SPLINE
SPL {X  -134.098, Y  +772.750, Z    +0.000, E1   -45.587, E3 +302845.435}
SPL {X  -155.319, Y  +733.085, Z    +0.000, E1   -31.947, E3 +302836.313}
SPL {X  -162.077, Y  +709.719, Z    +0.000, E1   -21.590, E3 +302837.990}
SPL {X  -164.499, Y  +694.994, Z    +0.000, E1   -13.860, E3 +302838.775}
SPL {X  -165.382, Y  +684.927, Z    +0.000, E1    -7.984, E3 +302836.952}
SPL {X  -165.645, Y  +676.778, Z    +0.000, E1    -2.777, E3 +302836.675}
SPL {X  -165.650, Y  +672.041, Z    +0.000, E1    +0.844, E3 +302835.366}
SPL {X  -165.650, Y  +667.328, Z    +0.000, E1    +5.806, E3 +302834.743}
SPL {X  -165.650, Y  +661.774, Z    +0.000, E1   +13.006, E3 +302833.067}
SPL {X  -165.650, Y  +656.573, Z    +0.000, E1   +19.875, E3 +302833.626}
SPL {X  -165.650, Y  +650.769, Z    +0.000, E1   +28.083, E3 +302831.992}
SPL {X  -165.650, Y  +639.700, Z    +0.000, E1   +43.326, E3 +302827.054}
SPL {X  -165.650, Y  +605.320, Z    +0.000, E1   +76.562, E3 +302806.463}
SPL {X  -165.650, Y  +597.745, Z    +0.000, E1   +59.636, E3 +302844.464}
SPL {X  -165.650, Y  +596.360, Z    +0.000, E1   +54.978, E3 +302858.072}
SPL {X  -165.650, Y  +524.050, Z    +0.000, E1   +59.300, E3 +302919.978}
ENDSPLINE

SPLINE
SPL {X  -165.650, Y  +539.856, Z    +0.000, E1   +53.398, E3 +302935.626}
ENDSPLINE

SPLINE
SPL {X  -165.650, Y  +530.389, Z    +0.000, E1   +53.621, E3 +302948.631}
SPL {X  -165.650, Y  +521.849, Z    +0.000, E1   +53.452, E3 +302962.571}
SPL {X  -165.650, Y  +515.134, Z    +0.000, E1   +53.252, E3 +302973.922}
SPL {X  -165.650, Y  +505.685, Z    +0.000, E1   +53.701, E3 +302985.529}
SPL {X  -165.650, Y  +498.275, Z    +0.000, E1   +53.357, E3 +302998.837}
SPL {X  -165.650, Y  +491.031, Z    +0.000, E1   +53.348, E3 +303009.857}
SPL {X  -165.650, Y  +479.077, Z    +0.000, E1   +55.039, E3 +303016.980}
SPL {X  -165.650, Y  +450.615, Z    +0.000, E1   +59.721, E3 +303023.486}
SPL {X  -165.650, Y  +449.326, Z    +0.000, E1   +58.606, E3 +303032.535}
SPL {X  -165.650, Y  +442.154, Z    +0.000, E1   +58.369, E3 +303043.159}
SPL {X  -165.650, Y  +437.405, Z    +0.000, E1   +57.663, E3 +303053.769}
SPL {X  -165.650, Y  +432.227, Z    +0.000, E1   +57.103, E3 +303064.256}
SPL {X  -165.650, Y  +428.683, Z    +0.000, E1   +56.222, E3 +303074.611}
SPL {X  -165.650, Y  +424.202, Z    +0.000, E1   +55.382, E3 +303086.300}
SPL {X  -165.650, Y  +418.756, Z    +0.000, E1   +54.154, E3 +303101.979}
SPL {X  -165.650, Y  +407.872, Z    +0.000, E1   +54.003, E3 +303119.064}
SPL {X  -165.650, Y  +400.791, Z    +0.000, E1   +53.827, E3 +303130.507}
SPL {X  -165.650, Y  +393.046, Z    +0.000, E1   +53.951, E3 +303141.399}
SPL {X  -165.650, Y  +383.306, Z    +0.000, E1   +53.987, E3 +303155.676}
SPL {X  -165.640, Y  +376.676, Z    +0.000, E1   +53.760, E3 +303166.843}
SPL {X  -165.408, Y  +369.556, Z    +0.000, E1   +53.942, E3 +303176.394}
SPL {X  -164.927, Y  +363.041, Z    +0.000, E1   +53.687, E3 +303187.690}
SPL {X  -164.096, Y  +355.862, Z    +0.000, E1   +53.838, E3 +303197.420}
SPL {X  -162.936, Y  +348.637, Z    +0.000, E1   +53.390, E3 +303211.136}
SPL {X  -161.218, Y  +340.437, Z    +0.000, E1   +53.207, E3 +303224.248}
SPL {X  -159.523, Y  +333.864, Z    +0.000, E1   +52.908, E3 +303235.870}
SPL {X  -157.624, Y  +327.563, Z    +0.000, E1   +52.705, E3 +303246.280}
SPL {X  -155.665, Y  +321.859, Z    +0.000, E1   +52.064, E3 +303258.453}
SPL {X  -152.682, Y  +314.249, Z    +0.000, E1   +51.841, E3 +303270.901}
SPL {X  -150.607, Y  +309.525, Z    +0.000, E1   +51.147, E3 +303281.385}
SPL {X  -142.104, Y  +293.374, Z    +0.000, E1   +55.775, E3 +303281.117}
SPL {X  -134.755, Y  +282.163, Z    +0.000, E1   +57.236, E3 +303287.385}
SPL {X  -117.053, Y  +261.289, Z    +0.000, E1   +49.815, E3 +303396.897}
ENDSPLINE

SPLINE
SPL {X  -148.836, Y  +305.783, Z    +0.000, E1   +38.029, E3 +303488.375}
SPL {X  -161.816, Y  +343.065, Z    +0.000, E1   +22.147, E3 +303479.025}
SPL {X  -164.614, Y  +360.007, Z    +0.000, E1   +13.213, E3 +303474.811}
SPL {X  -165.520, Y  +371.933, Z    +0.000, E1    +6.276, E3 +303477.565}
SPL {X  -165.650, Y  +378.704, Z    +0.000, E1    +1.700, E3 +303476.435}
SPL {X  -165.650, Y  +382.197, Z    +0.000, E1    -1.038, E3 +303475.508}
SPL {X  -165.650, Y  +386.782, Z    +0.000, E1    -5.783, E3 +303474.986}
SPL {X  -165.650, Y  +392.406, Z    +0.000, E1   -13.042, E3 +303472.883}
SPL {X  -165.650, Y  +398.038, Z    +0.000, E1   -20.113, E3 +303474.450}
SPL {X  -165.650, Y  +403.005, Z    +0.000, E1   -26.762, E3 +303473.632}
SPL {X  -165.650, Y  +415.469, Z    +0.000, E1   -43.461, E3 +303468.455}
SPL {X  -165.650, Y  +460.095, Z    +0.000, E1   -60.221, E3 +303486.717}
SPL {X  -165.650, Y  +535.749, Z    +0.000, E1   -60.559, E3 +303557.560}
ENDSPLINE

SPLINE
SPL {X  -165.650, Y  +516.750, Z    +0.000, E1   -54.244, E3 +303573.411}
ENDSPLINE

SPLINE
SPL {X  -165.650, Y  +524.345, Z    +0.000, E1   -54.115, E3 +303585.308}
SPL {X  -165.650, Y  +531.171, Z    +0.000, E1   -54.075, E3 +303595.746}
SPL {X  -165.650, Y  +538.771, Z    +0.000, E1   -53.840, E3 +303608.486}
SPL {X  -165.650, Y  +548.103, Z    +0.000, E1   -53.944, E3 +303621.833}
SPL {X  -165.650, Y  +558.071, Z    +0.000, E1   -53.870, E3 +303637.174}
SPL {X  -165.650, Y  +568.053, Z    +0.000, E1   -54.124, E3 +303650.351}
SPL {X  -165.650, Y  +577.021, Z    +0.000, E1   -53.813, E3 +303665.850}
SPL {X  -165.650, Y  +587.996, Z    +0.000, E1   -53.969, E3 +303681.088}
SPL {X  -165.650, Y  +595.185, Z    +0.000, E1   -53.962, E3 +303691.797}
SPL {X  -165.650, Y  +602.138, Z    +0.000, E1   -53.941, E3 +303702.291}
SPL {X  -165.650, Y  +610.307, Z    +0.000, E1   -53.995, E3 +303714.139}
SPL {X  -165.650, Y  +617.878, Z    +0.000, E1   -53.838, E3 +303726.396}
SPL {X  -165.650, Y  +626.374, Z    +0.000, E1   -54.092, E3 +303737.411}
SPL {X  -165.650, Y  +632.964, Z    +0.000, E1   -53.887, E3 +303748.539}
SPL {X  -165.650, Y  +640.262, Z    +0.000, E1   -53.965, E3 +303758.853}
SPL {X  -165.650, Y  +647.911, Z    +0.000, E1   -53.930, E3 +303770.608}
SPL {X  -165.650, Y  +658.189, Z    +0.000, E1   -53.932, E3 +303785.908}
SPL {X  -165.650, Y  +667.820, Z    +0.000, E1   -53.975, E3 +303799.934}
SPL {X  -165.623, Y  +678.503, Z    +0.000, E1   -53.932, E3 +303816.286}
SPL {X  -165.171, Y  +688.090, Z    +0.000, E1   -54.025, E3 +303829.734}
SPL {X  -164.558, Y  +694.489, Z    +0.000, E1   -53.745, E3 +303841.083}
SPL {X  -163.580, Y  +701.606, Z    +0.000, E1   -53.591, E3 +303852.516}
SPL {X  -162.702, Y  +706.614, Z    +0.000, E1   -53.230, E3 +303862.183}
SPL {X  -160.941, Y  +714.715, Z    +0.000, E1   -53.321, E3 +303873.802}
SPL {X  -159.638, Y  +719.723, Z    +0.000, E1   -52.685, E3 +303884.805}
SPL {X  -157.521, Y  +726.754, Z    +0.000, E1   -52.585, E3 +303896.000}
SPL {X  -155.632, Y  +732.234, Z    +0.000, E1   -52.209, E3 +303906.047}
SPL {X  -153.975, Y  +736.588, Z    +0.000, E1   -51.877, E3 +303914.373}
SPL {X  -151.949, Y  +741.465, Z    +0.000, E1   -51.645, E3 +303922.779}
SPL {X  -149.075, Y  +747.727, Z    +0.000, E1   -52.134, E3 +303929.493}
SPL {X  -137.775, Y  +767.467, Z    +0.000, E1   -56.912, E3 +303932.157}
SPL {X  -128.847, Y  +779.607, Z    +0.000, E1   -49.118, E3 +304007.173}
SPL {X   -94.133, Y  +811.804, Z    +0.000, E1   -53.019, E3 +304061.807}
ENDSPLINE

SPLINE
SPL {X  -123.886, Y  +785.464, Z    +0.000, E1   -49.465, E3 +304146.834}
SPL {X  -152.385, Y  +740.452, Z    +0.000, E1   -34.821, E3 +304127.811}
SPL {X  -162.077, Y  +709.719, Z    +0.000, E1   -21.590, E3 +304129.657}
SPL {X  -164.499, Y  +694.994, Z    +0.000, E1   -13.860, E3 +304130.442}
SPL {X  -165.382, Y  +684.927, Z    +0.000, E1    -7.984, E3 +304128.619}
SPL {X  -165.645, Y  +676.778, Z    +0.000, E1    -2.777, E3 +304128.341}
SPL {X  -165.650, Y  +672.041, Z    +0.000, E1    +0.844, E3 +304127.033}
SPL {X  -165.650, Y  +667.328, Z    +0.000, E1    +5.806, E3 +304126.410}
SPL {X  -165.650, Y  +661.774, Z    +0.000, E1   +13.006, E3 +304124.734}
SPL {X  -165.650, Y  +654.085, Z    +0.000, E1   +23.232, E3 +304124.593}
SPL {X  -165.650, Y  +639.700, Z    +0.000, E1   +43.326, E3 +304118.720}
SPL {X  -165.650, Y  +605.320, Z    +0.000, E1   +76.562, E3 +304098.130}
SPL {X  -165.650, Y  +597.745, Z    +0.000, E1   +59.636, E3 +304136.131}
SPL {X  -165.650, Y  +596.360, Z    +0.000, E1   +54.978, E3 +304149.739}
SPL {X  -165.650, Y  +524.050, Z    +0.000, E1   +59.300, E3 +304211.645}
ENDSPLINE

SPLINE
SPL {X  -165.650, Y  +539.856, Z    +0.000, E1   +53.398, E3 +304227.292}
ENDSPLINE

SPLINE
SPL {X  -165.650, Y  +530.389, Z    +0.000, E1   +53.621, E3 +304240.298}
SPL {X  -165.650, Y  +521.849, Z    +0.000, E1   +53.452, E3 +304254.237}
SPL {X  -165.650, Y  +515.134, Z    +0.000, E1   +53.252, E3 +304265.588}
SPL {X  -165.650, Y  +505.685, Z    +0.000, E1   +53.701, E3 +304277.196}
SPL {X  -165.650, Y  +498.275, Z    +0.000, E1   +53.357, E3 +304290.504}
SPL {X  -165.650, Y  +491.031, Z    +0.000, E1   +53.348, E3 +304301.524}
SPL {X  -165.650, Y  +479.077, Z    +0.000, E1   +55.039, E3 +304308.647}
SPL {X  -165.650, Y  +450.615, Z    +0.000, E1   +59.721, E3 +304315.152}
SPL {X  -165.650, Y  +449.326, Z    +0.000, E1   +58.606, E3 +304324.202}
SPL {X  -165.650, Y  +442.154, Z    +0.000, E1   +58.369, E3 +304334.826}
SPL {X  -165.650, Y  +437.405, Z    +0.000, E1   +57.663, E3 +304345.435}
SPL {X  -165.650, Y  +432.227, Z    +0.000, E1   +57.103, E3 +304355.923}
SPL {X  -165.650, Y  +428.683, Z    +0.000, E1   +56.222, E3 +304366.277}
SPL {X  -165.650, Y  +424.202, Z    +0.000, E1   +55.382, E3 +304377.966}
SPL {X  -165.650, Y  +420.516, Z    +0.000, E1   +54.144, E3 +304390.972}
ENDSPLINE

SPLINE
SPL {X  -165.650, Y  +429.698, Z    +0.000, E1   +49.459, E3 +304404.987}
ENDSPLINE

SPLINE
SPL {X  -165.650, Y  +421.000, Z    +0.000, E1   +49.266, E3 +304421.417}
SPL {X  -165.650, Y  +412.094, Z    +0.000, E1   +49.264, E3 +304437.104}
SPL {X  -165.650, Y  +402.476, Z    +0.000, E1   +49.356, E3 +304453.521}
SPL {X  -165.650, Y  +393.708, Z    +0.000, E1   +49.252, E3 +304469.512}
SPL {X  -165.650, Y  +386.526, Z    +0.000, E1   +49.193, E3 +304482.457}
SPL {X  -165.649, Y  +378.059, Z    +0.000, E1   +49.283, E3 +304497.000}
SPL {X  -165.370, Y  +368.879, Z    +0.000, E1   +49.286, E3 +304513.081}
SPL {X  -164.828, Y  +362.023, Z    +0.000, E1   +48.964, E3 +304527.042}
SPL {X  -163.908, Y  +354.543, Z    +0.000, E1   +49.169, E3 +304538.990}
SPL {X  -163.052, Y  +349.277, Z    +0.000, E1   +48.680, E3 +304551.095}
SPL {X  -162.125, Y  +344.507, Z    +0.000, E1   +48.543, E3 +304560.235}
SPL {X  -160.947, Y  +339.310, Z    +0.000, E1   +48.561, E3 +304569.344}
SPL {X  -159.499, Y  +333.778, Z    +0.000, E1   +48.145, E3 +304581.456}
SPL {X  -157.380, Y  +326.814, Z    +0.000, E1   +47.797, E3 +304595.728}
SPL {X  -155.465, Y  +321.311, Z    +0.000, E1   +47.446, E3 +304607.106}
SPL {X  -153.706, Y  +316.739, Z    +0.000, E1   +47.523, E3 +304614.719}
SPL {X  -143.727, Y  +296.145, Z    +0.000, E1   +53.260, E3 +304617.863}
SPL {X  -128.440, Y  +273.891, Z    +0.000, E1   +47.966, E3 +304705.109}
ENDSPLINE

SPLINE
SPL {X  -131.798, Y  +278.155, Z    +0.000, E1   +45.574, E3 +304730.736}
SPL {X  -154.181, Y  +317.936, Z    +0.000, E1   +32.662, E3 +304796.072}
SPL {X  -162.537, Y  +346.536, Z    +0.000, E1   +20.123, E3 +304795.293}
SPL {X  -164.610, Y  +359.970, Z    +0.000, E1   +13.118, E3 +304790.159}
SPL {X  -165.367, Y  +368.828, Z    +0.000, E1    +8.137, E3 +304788.612}
SPL {X  -165.621, Y  +375.422, Z    +0.000, E1    +4.067, E3 +304789.489}
SPL {X  -165.650, Y  +379.733, Z    +0.000, E1    +1.160, E3 +304787.795}
SPL {X  -165.650, Y  +383.552, Z    +0.000, E1    -1.868, E3 +304787.045}
SPL {X  -165.650, Y  +387.323, Z    +0.000, E1    -5.609, E3 +304786.861}
SPL {X  -165.650, Y  +392.013, Z    +0.000, E1   -10.856, E3 +304785.878}
SPL {X  -165.650, Y  +398.769, Z    +0.000, E1   -19.304, E3 +304784.490}
SPL {X  -165.650, Y  +410.885, Z    +0.000, E1   -34.864, E3 +304780.166}
SPL {X  -165.650, Y  +446.037, Z    +0.000, E1   -53.739, E3 +304794.230}
SPL {X  -165.650, Y  +454.158, Z    +0.000, E1   -53.343, E3 +304804.582}
SPL {X  -165.650, Y  +513.780, Z    +0.000, E1   -56.183, E3 +304865.379}
ENDSPLINE

SPLINE
SPL {X  -165.650, Y  +495.869, Z    +0.000, E1   -48.812, E3 +304881.567}
ENDSPLINE

SPLINE
SPL {X  -165.650, Y  +504.906, Z    +0.000, E1   -48.979, E3 +304896.887}
SPL {X  -165.650, Y  +512.952, Z    +0.000, E1   -48.898, E3 +304911.509}
SPL {X  -165.650, Y  +519.321, Z    +0.000, E1   -49.041, E3 +304921.977}
SPL {X  -165.650, Y  +524.312, Z    +0.000, E1   -48.855, E3 +304932.002}
SPL {X  -165.650, Y  +530.631, Z    +0.000, E1   -48.990, E3 +304942.462}
SPL {X  -165.650, Y  +536.725, Z    +0.000, E1   -48.843, E3 +304954.213}
SPL {X  -165.650, Y  +542.959, Z    +0.000, E1   -48.923, E3 +304964.828}
SPL {X  -165.650, Y  +548.939, Z    +0.000, E1   -48.968, E3 +304975.222}
SPL {X  -165.650, Y  +553.607, Z    +0.000, E1   -48.716, E3 +304985.040}
SPL {X  -165.650, Y  +560.535, Z    +0.000, E1   -49.121, E3 +304994.988}
SPL {X  -165.650, Y  +564.320, Z    +0.000, E1   -48.789, E3 +305003.676}
SPL {X  -165.650, Y  +570.317, Z    +0.000, E1   -48.893, E3 +305013.843}
SPL {X  -165.650, Y  +577.487, Z    +0.000, E1   -49.001, E3 +305025.951}
SPL {X  -165.650, Y  +581.837, Z    +0.000, E1   -48.612, E3 +305035.984}
SPL {X  -165.650, Y  +588.614, Z    +0.000, E1   -49.053, E3 +305045.502}
SPL {X  -165.650, Y  +593.784, Z    +0.000, E1   -48.711, E3 +305056.787}
SPL {X  -165.650, Y  +600.281, Z    +0.000, E1   -48.957, E3 +305066.890}
SPL {X  -165.650, Y  +606.252, Z    +0.000, E1   -48.984, E3 +305077.423}
SPL {X  -165.650, Y  +612.690, Z    +0.000, E1   -49.044, E3 +305088.452}
SPL {X  -165.650, Y  +617.274, Z    +0.000, E1   -48.670, E3 +305098.901}
SPL {X  -165.650, Y  +624.267, Z    +0.000, E1   -48.953, E3 +305109.713}
SPL {X  -165.650, Y  +630.315, Z    +0.000, E1   -49.009, E3 +305120.143}
SPL {X  -165.650, Y  +635.030, Z    +0.000, E1   -48.821, E3 +305129.628}
SPL {X  -165.650, Y  +641.084, Z    +0.000, E1   -48.892, E3 +305140.110}
SPL {X  -165.650, Y  +648.143, Z    +0.000, E1   -49.033, E3 +305151.779}
SPL {X  -165.650, Y  +655.847, Z    +0.000, E1   -48.917, E3 +305166.397}
SPL {X  -165.650, Y  +663.676, Z    +0.000, E1   -48.809, E3 +305180.835}
SPL {X  -165.650, Y  +669.580, Z    +0.000, E1   -48.844, E3 +305191.173}
SPL {X  -165.650, Y  +675.734, Z    +0.000, E1   -49.021, E3 +305201.079}
SPL {X  -165.552, Y  +681.198, Z    +0.000, E1   -48.804, E3 +305212.160}
SPL {X  -165.221, Y  +687.413, Z    +0.000, E1   -48.790, E3 +305223.331}
SPL {X  -164.785, Y  +692.407, Z    +0.000, E1   -48.653, E3 +305233.047}
SPL {X  -164.074, Y  +698.293, Z    +0.000, E1   -48.857, E3 +305242.331}
SPL {X  -163.489, Y  +702.172, Z    +0.000, E1   -48.443, E3 +305251.648}
SPL {X  -162.671, Y  +706.776, Z    +0.000, E1   -48.273, E3 +305260.867}
SPL {X  -161.177, Y  +713.734, Z    +0.000, E1   -48.156, E3 +305274.153}
SPL {X  -159.392, Y  +720.602, Z    +0.000, E1   -47.892, E3 +305287.707}
SPL {X  -157.947, Y  +725.428, Z    +0.000, E1   -47.498, E3 +305298.446}
SPL {X  -155.696, Y  +732.057, Z    +0.000, E1   -47.224, E3 +305311.923}
SPL {X  -152.475, Y  +740.240, Z    +0.000, E1   -48.059, E3 +305321.752}
SPL {X  -143.211, Y  +758.749, Z    +0.000, E1   -53.445, E3 +305322.793}
SPL {X  -129.526, Y  +778.761, Z    +0.000, E1   -47.396, E3 +305413.535}
ENDSPLINE

SPLINE
SPL {X  -152.848, Y  +739.355, Z    +0.000, E1   -33.672, E3 +305489.104}
SPL {X  -162.700, Y  +706.622, Z    +0.000, E1   -19.657, E3 +305495.260}
SPL {X  -164.822, Y  +692.043, Z    +0.000, E1   -12.043, E3 +305490.899}
SPL {X  -165.501, Y  +682.513, Z    +0.000, E1    -6.586, E3 +305489.593}
SPL {X  -165.650, Y  +674.436, Z    +0.000, E1    -1.443, E3 +305488.369}
SPL {X  -165.650, Y  +669.008, Z    +0.000, E1    +2.993, E3 +305487.924}
SPL {X  -165.650, Y  +664.048, Z    +0.000, E1    +8.230, E3 +305487.203}
SPL {X  -165.650, Y  +658.867, Z    +0.000, E1   +14.313, E3 +305485.666}
SPL {X  -165.650, Y  +650.683, Z    +0.000, E1   +24.801, E3 +305483.102}
SPL {X  -165.650, Y  +636.402, Z    +0.000, E1   +39.824, E3 +305483.065}
SPL {X  -165.650, Y  +586.376, Z    +0.000, E1   +59.481, E3 +305500.737}
SPL {X  -165.650, Y  +536.483, Z    +0.000, E1   +57.139, E3 +305562.506}
ENDSPLINE

SPLINE
SPL {X  -165.650, Y  +561.248, Z    +0.000, E1   +49.247, E3 +305573.196}
ENDSPLINE

SPLINE
SPL {X  -165.650, Y  +558.330, Z    +0.000, E1   +47.867, E3 +305586.920}
SPL {X  -165.650, Y  +549.545, Z    +0.000, E1   +47.953, E3 +305602.592}
SPL {X  -165.650, Y  +541.974, Z    +0.000, E1   +47.882, E3 +305616.981}
SPL {X  -165.650, Y  +535.023, Z    +0.000, E1   +47.697, E3 +305630.970}
SPL {X  -165.650, Y  +526.169, Z    +0.000, E1   +47.853, E3 +305646.565}
SPL {X  -165.650, Y  +517.493, Z    +0.000, E1   +47.895, E3 +305662.312}
SPL {X  -165.650, Y  +511.255, Z    +0.000, E1   +47.920, E3 +305673.601}
SPL {X  -165.650, Y  +507.257, Z    +0.000, E1   +47.748, E3 +305681.983}
SPL {X  -165.650, Y  +501.812, Z    +0.000, E1   +47.738, E3 +305692.266}
SPL {X  -165.650, Y  +493.465, Z    +0.000, E1   +47.959, E3 +305706.437}
SPL {X  -165.650, Y  +486.149, Z    +0.000, E1   +47.831, E3 +305720.712}
SPL {X  -165.650, Y  +479.821, Z    +0.000, E1   +47.727, E3 +305732.985}
SPL {X  -165.650, Y  +472.739, Z    +0.000, E1   +47.923, E3 +305745.005}
SPL {X  -165.650, Y  +465.366, Z    +0.000, E1   +47.775, E3 +305759.584}
SPL {X  -165.650, Y  +457.811, Z    +0.000, E1   +47.987, E3 +305772.201}
SPL {X  -165.650, Y  +451.187, Z    +0.000, E1   +47.917, E3 +305784.945}
SPL {X  -165.650, Y  +439.019, Z    +0.000, E1   +49.830, E3 +305795.267}
SPL {X  -165.650, Y  +435.473, Z    +0.000, E1   +49.263, E3 +305804.988}
SPL {X  -165.650, Y  +428.379, Z    +0.000, E1   +49.373, E3 +305816.760}
SPL {X  -165.650, Y  +423.272, Z    +0.000, E1   +49.176, E3 +305826.896}
SPL {X  -165.650, Y  +416.522, Z    +0.000, E1   +49.338, E3 +305837.874}
SPL {X  -165.650, Y  +410.777, Z    +0.000, E1   +49.173, E3 +305848.926}
SPL {X  -165.650, Y  +402.476, Z    +0.000, E1   +49.356, E3 +305862.612}
SPL {X  -165.650, Y  +393.708, Z    +0.000, E1   +49.252, E3 +305878.602}
SPL {X  -165.650, Y  +386.526, Z    +0.000, E1   +49.193, E3 +305891.548}
SPL {X  -165.650, Y  +381.684, Z    +0.000, E1   +49.061, E3 +305900.833}
SPL {X  -165.602, Y  +374.507, Z    +0.000, E1   +49.269, E3 +305912.425}
SPL {X  -165.255, Y  +367.073, Z    +0.000, E1   +49.394, E3 +305924.617}
SPL {X  -164.828, Y  +362.023, Z    +0.000, E1   +48.964, E3 +305936.133}
SPL {X  -163.908, Y  +354.543, Z    +0.000, E1   +49.169, E3 +305948.081}
SPL {X  -163.052, Y  +349.277, Z    +0.000, E1   +48.680, E3 +305960.186}
SPL {X  -162.125, Y  +344.507, Z    +0.000, E1   +48.543, E3 +305969.326}
SPL {X  -160.947, Y  +339.310, Z    +0.000, E1   +48.561, E3 +305978.435}
SPL {X  -159.860, Y  +335.086, Z    +0.000, E1   +48.145, E3 +305988.147}
SPL {X  -158.277, Y  +329.631, Z    +0.000, E1   +47.981, E3 +305998.769}
SPL {X  -156.804, Y  +325.092, Z    +0.000, E1   +47.609, E3 +306008.662}
SPL {X  -155.465, Y  +321.311, Z    +0.000, E1   +47.446, E3 +306016.197}
SPL {X  -153.706, Y  +316.739, Z    +0.000, E1   +47.523, E3 +306023.810}
SPL {X  -143.727, Y  +296.145, Z    +0.000, E1   +53.260, E3 +306026.954}
SPL {X  -128.440, Y  +273.891, Z    +0.000, E1   +47.966, E3 +306114.200}
ENDSPLINE

SPLINE
SPL {X  -131.798, Y  +278.155, Z    +0.000, E1   +45.574, E3 +306139.827}
SPL {X  -154.181, Y  +317.936, Z    +0.000, E1   +32.662, E3 +306205.163}
SPL {X  -162.537, Y  +346.536, Z    +0.000, E1   +20.123, E3 +306204.384}
SPL {X  -164.610, Y  +359.970, Z    +0.000, E1   +13.118, E3 +306199.250}
SPL {X  -165.367, Y  +368.828, Z    +0.000, E1    +8.137, E3 +306197.703}
SPL {X  -165.621, Y  +375.422, Z    +0.000, E1    +4.067, E3 +306198.580}
SPL {X  -165.650, Y  +379.733, Z    +0.000, E1    +1.160, E3 +306196.886}
SPL {X  -165.650, Y  +383.552, Z    +0.000, E1    -1.868, E3 +306196.135}
SPL {X  -165.650, Y  +387.323, Z    +0.000, E1    -5.609, E3 +306195.952}
SPL {X  -165.650, Y  +392.013, Z    +0.000, E1   -10.856, E3 +306194.969}
SPL {X  -165.650, Y  +398.769, Z    +0.000, E1   -19.304, E3 +306193.580}
SPL {X  -165.650, Y  +410.885, Z    +0.000, E1   -34.864, E3 +306189.257}
SPL {X  -165.650, Y  +448.279, Z    +0.000, E1   -53.294, E3 +306207.102}
SPL {X  -165.650, Y  +465.286, Z    +0.000, E1   -55.209, E3 +306220.953}
SPL {X  -165.650, Y  +513.874, Z    +0.000, E1   -57.683, E3 +306265.762}
ENDSPLINE

SPLINE
SPL {X  -165.650, Y  +513.412, Z    +0.000, E1   -55.245, E3 +306279.357}
SPL {X  -165.650, Y  +495.869, Z    +0.000, E1   -48.812, E3 +306290.658}
ENDSPLINE

SPLINE
SPL {X  -165.650, Y  +502.040, Z    +0.000, E1   -48.856, E3 +306301.402}
SPL {X  -165.650, Y  +507.863, Z    +0.000, E1   -49.013, E3 +306310.822}
SPL {X  -165.650, Y  +512.952, Z    +0.000, E1   -48.898, E3 +306320.599}
SPL {X  -165.650, Y  +519.321, Z    +0.000, E1   -49.041, E3 +306331.067}
SPL {X  -165.650, Y  +524.312, Z    +0.000, E1   -48.855, E3 +306341.093}
SPL {X  -165.650, Y  +530.631, Z    +0.000, E1   -48.990, E3 +306351.553}
SPL {X  -165.650, Y  +536.725, Z    +0.000, E1   -48.843, E3 +306363.304}
SPL {X  -165.650, Y  +542.959, Z    +0.000, E1   -48.923, E3 +306373.919}
SPL {X  -165.650, Y  +548.939, Z    +0.000, E1   -48.968, E3 +306384.312}
SPL {X  -165.650, Y  +553.607, Z    +0.000, E1   -48.716, E3 +306394.130}
SPL {X  -165.650, Y  +560.535, Z    +0.000, E1   -49.121, E3 +306404.079}
SPL {X  -165.650, Y  +564.320, Z    +0.000, E1   -48.789, E3 +306412.767}
SPL {X  -165.650, Y  +570.317, Z    +0.000, E1   -48.893, E3 +306422.933}
SPL {X  -165.650, Y  +577.487, Z    +0.000, E1   -49.001, E3 +306435.042}
SPL {X  -165.650, Y  +581.837, Z    +0.000, E1   -48.612, E3 +306445.075}
SPL {X  -165.650, Y  +588.614, Z    +0.000, E1   -49.053, E3 +306454.593}
SPL {X  -165.650, Y  +593.784, Z    +0.000, E1   -48.711, E3 +306465.878}
SPL {X  -165.650, Y  +600.281, Z    +0.000, E1   -48.957, E3 +306475.981}
SPL {X  -165.650, Y  +606.252, Z    +0.000, E1   -48.984, E3 +306486.514}
SPL {X  -165.650, Y  +612.690, Z    +0.000, E1   -49.044, E3 +306497.543}
SPL {X  -165.650, Y  +617.274, Z    +0.000, E1   -48.670, E3 +306507.992}
SPL {X  -165.650, Y  +624.267, Z    +0.000, E1   -48.953, E3 +306518.804}
SPL {X  -165.650, Y  +632.510, Z    +0.000, E1   -48.976, E3 +306533.558}
SPL {X  -165.650, Y  +641.084, Z    +0.000, E1   -48.892, E3 +306549.201}
SPL {X  -165.650, Y  +648.143, Z    +0.000, E1   -49.033, E3 +306560.870}
SPL {X  -165.650, Y  +655.847, Z    +0.000, E1   -48.917, E3 +306575.488}
SPL {X  -165.650, Y  +663.676, Z    +0.000, E1   -48.809, E3 +306589.925}
SPL {X  -165.650, Y  +669.580, Z    +0.000, E1   -48.844, E3 +306600.264}
SPL {X  -165.650, Y  +675.734, Z    +0.000, E1   -49.021, E3 +306610.170}
SPL {X  -165.552, Y  +681.198, Z    +0.000, E1   -48.804, E3 +306621.251}
SPL {X  -165.221, Y  +687.413, Z    +0.000, E1   -48.790, E3 +306632.422}
SPL {X  -164.785, Y  +692.407, Z    +0.000, E1   -48.653, E3 +306642.138}
SPL {X  -164.074, Y  +698.293, Z    +0.000, E1   -48.857, E3 +306651.422}
SPL {X  -163.489, Y  +702.172, Z    +0.000, E1   -48.443, E3 +306660.739}
SPL {X  -162.217, Y  +709.048, Z    +0.000, E1   -48.328, E3 +306673.878}
SPL {X  -160.800, Y  +715.289, Z    +0.000, E1   -47.964, E3 +306686.886}
SPL {X  -159.392, Y  +720.602, Z    +0.000, E1   -47.892, E3 +306696.798}
SPL {X  -157.947, Y  +725.428, Z    +0.000, E1   -47.498, E3 +306707.537}
SPL {X  -156.133, Y  +730.838, Z    +0.000, E1   -47.305, E3 +306718.254}
SPL {X  -154.870, Y  +734.280, Z    +0.000, E1   -46.924, E3 +306726.257}
SPL {X  -150.529, Y  +744.645, Z    +0.000, E1   -49.720, E3 +306729.531}
SPL {X  -140.987, Y  +762.463, Z    +0.000, E1   -53.922, E3 +306734.562}
SPL {X  -129.526, Y  +778.761, Z    +0.000, E1   -47.396, E3 +306822.626}
ENDSPLINE

SPLINE
SPL {X  -152.848, Y  +739.355, Z    +0.000, E1   -33.672, E3 +306898.195}
SPL {X  -162.700, Y  +706.622, Z    +0.000, E1   -19.657, E3 +306904.351}
SPL {X  -164.822, Y  +692.043, Z    +0.000, E1   -12.043, E3 +306899.990}
SPL {X  -165.501, Y  +682.513, Z    +0.000, E1    -6.586, E3 +306898.684}
SPL {X  -165.645, Y  +676.829, Z    +0.000, E1    -2.974, E3 +306898.028}
SPL {X  -165.650, Y  +673.338, Z    +0.000, E1    -0.547, E3 +306897.197}
SPL {X  -165.650, Y  +669.008, Z    +0.000, E1    +2.993, E3 +306897.015}
SPL {X  -165.650, Y  +663.208, Z    +0.000, E1    +9.118, E3 +306896.099}
SPL {X  -165.650, Y  +657.399, Z    +0.000, E1   +16.251, E3 +306894.218}
SPL {X  -165.650, Y  +650.683, Z    +0.000, E1   +24.801, E3 +306892.193}
SPL {X  -165.650, Y  +636.402, Z    +0.000, E1   +39.824, E3 +306892.155}
SPL {X  -165.650, Y  +586.376, Z    +0.000, E1   +59.481, E3 +306909.828}
SPL {X  -165.650, Y  +558.853, Z    +0.000, E1   +50.142, E3 +306981.298}
SPL {X  -165.650, Y  +558.330, Z    +0.000, E1   +47.867, E3 +306996.011}
SPL {X  -165.650, Y  +549.545, Z    +0.000, E1   +47.953, E3 +307011.683}
SPL {X  -165.650, Y  +544.306, Z    +0.000, E1   +47.619, E3 +307023.241}
SPL {X  -165.650, Y  +537.837, Z    +0.000, E1   +47.880, E3 +307033.767}
SPL {X  -165.650, Y  +530.616, Z    +0.000, E1   +47.886, E3 +307047.132}
SPL {X  -165.650, Y  +522.460, Z    +0.000, E1   +47.738, E3 +307063.242}
SPL {X  -165.650, Y  +512.416, Z    +0.000, E1   +48.035, E3 +307080.007}
SPL {X  -165.650, Y  +507.257, Z    +0.000, E1   +47.748, E3 +307091.074}
SPL {X  -165.650, Y  +501.812, Z    +0.000, E1   +47.738, E3 +307101.357}
SPL {X  -165.650, Y  +494.522, Z    +0.000, E1   +48.055, E3 +307112.884}
SPL {X  -165.650, Y  +489.529, Z    +0.000, E1   +47.849, E3 +307123.338}
SPL {X  -165.650, Y  +481.894, Z    +0.000, E1   +47.756, E3 +307138.239}
SPL {X  -165.650, Y  +472.739, Z    +0.000, E1   +47.923, E3 +307154.096}
SPL {X  -165.650, Y  +465.366, Z    +0.000, E1   +47.775, E3 +307168.675}
SPL {X  -165.650, Y  +456.851, Z    +0.000, E1   +47.856, E3 +307183.982}
SPL {X  -165.650, Y  +445.317, Z    +0.000, E1   +48.773, E3 +307199.560}
SPL {X  -165.650, Y  +435.473, Z    +0.000, E1   +49.263, E3 +307214.079}
SPL {X  -165.650, Y  +428.379, Z    +0.000, E1   +49.373, E3 +307225.851}
SPL {X  -165.650, Y  +421.000, Z    +0.000, E1   +49.266, E3 +307239.599}
SPL {X  -165.650, Y  +412.094, Z    +0.000, E1   +49.264, E3 +307255.286}
SPL {X  -165.650, Y  +402.476, Z    +0.000, E1   +49.356, E3 +307271.703}
SPL {X  -165.650, Y  +393.708, Z    +0.000, E1   +49.252, E3 +307287.693}
SPL {X  -165.650, Y  +386.526, Z    +0.000, E1   +49.193, E3 +307300.639}
SPL {X  -165.649, Y  +378.059, Z    +0.000, E1   +49.283, E3 +307315.182}
SPL {X  -165.370, Y  +368.879, Z    +0.000, E1   +49.286, E3 +307331.263}
SPL {X  -164.828, Y  +362.023, Z    +0.000, E1   +48.964, E3 +307345.224}
SPL {X  -163.908, Y  +354.543, Z    +0.000, E1   +49.169, E3 +307357.171}
SPL {X  -163.052, Y  +349.277, Z    +0.000, E1   +48.680, E3 +307369.277}
SPL {X  -162.125, Y  +344.507, Z    +0.000, E1   +48.543, E3 +307378.417}
SPL {X  -160.947, Y  +339.310, Z    +0.000, E1   +48.561, E3 +307387.526}
SPL {X  -159.499, Y  +333.778, Z    +0.000, E1   +48.145, E3 +307399.638}
SPL {X  -157.957, Y  +328.606, Z    +0.000, E1   +47.890, E3 +307410.063}
SPL {X  -156.095, Y  +323.055, Z    +0.000, E1   +47.566, E3 +307421.747}
SPL {X  -153.706, Y  +316.739, Z    +0.000, E1   +47.523, E3 +307432.901}
SPL {X  -143.727, Y  +296.145, Z    +0.000, E1   +53.260, E3 +307436.045}
SPL {X  -128.440, Y  +273.891, Z    +0.000, E1   +47.966, E3 +307523.291}
ENDSPLINE

SPLINE
SPL {X  -131.798, Y  +278.155, Z    +0.000, E1   +45.574, E3 +307548.918}
SPL {X  -154.181, Y  +317.936, Z    +0.000, E1   +32.662, E3 +307614.254}
SPL {X  -162.537, Y  +346.536, Z    +0.000, E1   +20.123, E3 +307613.475}
SPL {X  -164.610, Y  +359.970, Z    +0.000, E1   +13.118, E3 +307608.341}
SPL {X  -165.367, Y  +368.828, Z    +0.000, E1    +8.137, E3 +307606.794}
SPL {X  -165.621, Y  +375.422, Z    +0.000, E1    +4.067, E3 +307607.671}
SPL {X  -165.650, Y  +380.991, Z    +0.000, E1    +0.306, E3 +307605.682}
SPL {X  -165.650, Y  +384.571, Z    +0.000, E1    -2.883, E3 +307605.121}
SPL {X  -165.650, Y  +388.716, Z    +0.000, E1    -7.003, E3 +307604.631}
SPL {X  -165.650, Y  +396.644, Z    +0.000, E1   -16.434, E3 +307603.250}
SPL {X  -165.650, Y  +410.885, Z    +0.000, E1   -34.864, E3 +307598.348}
SPL {X  -165.650, Y  +446.037, Z    +0.000, E1   -53.739, E3 +307612.412}
SPL {X  -165.650, Y  +454.158, Z    +0.000, E1   -53.343, E3 +307622.764}
SPL {X  -165.650, Y  +513.780, Z    +0.000, E1   -56.183, E3 +307683.561}
ENDSPLINE

SPLINE
SPL {X  -165.650, Y  +495.869, Z    +0.000, E1   -48.812, E3 +307699.749}
ENDSPLINE

SPLINE
SPL {X  -165.650, Y  +502.040, Z    +0.000, E1   -48.856, E3 +307710.493}
SPL {X  -165.650, Y  +507.863, Z    +0.000, E1   -49.013, E3 +307719.913}
SPL {X  -165.650, Y  +512.952, Z    +0.000, E1   -48.898, E3 +307729.690}
SPL {X  -165.650, Y  +519.321, Z    +0.000, E1   -49.041, E3 +307740.158}
SPL {X  -165.650, Y  +524.312, Z    +0.000, E1   -48.855, E3 +307750.184}
SPL {X  -165.650, Y  +532.191, Z    +0.000, E1   -48.944, E3 +307763.852}
SPL {X  -165.650, Y  +541.400, Z    +0.000, E1   -48.945, E3 +307780.226}
SPL {X  -165.650, Y  +548.939, Z    +0.000, E1   -48.968, E3 +307793.403}
SPL {X  -165.650, Y  +553.607, Z    +0.000, E1   -48.716, E3 +307803.221}
SPL {X  -165.650, Y  +562.368, Z    +0.000, E1   -49.014, E3 +307817.282}
SPL {X  -165.650, Y  +570.317, Z    +0.000, E1   -48.893, E3 +307832.024}
SPL {X  -165.650, Y  +577.487, Z    +0.000, E1   -49.001, E3 +307844.132}
SPL {X  -165.650, Y  +581.837, Z    +0.000, E1   -48.612, E3 +307854.166}
SPL {X  -165.650, Y  +588.614, Z    +0.000, E1   -49.053, E3 +307863.684}
SPL {X  -165.650, Y  +593.784, Z    +0.000, E1   -48.711, E3 +307874.969}
SPL {X  -165.650, Y  +600.281, Z    +0.000, E1   -48.957, E3 +307885.072}
SPL {X  -165.650, Y  +606.252, Z    +0.000, E1   -48.984, E3 +307895.605}
SPL {X  -165.650, Y  +612.690, Z    +0.000, E1   -49.044, E3 +307906.634}
SPL {X  -165.650, Y  +617.274, Z    +0.000, E1   -48.670, E3 +307917.083}
SPL {X  -165.650, Y  +624.267, Z    +0.000, E1   -48.953, E3 +307927.895}
SPL {X  -165.650, Y  +630.315, Z    +0.000, E1   -49.009, E3 +307938.325}
SPL {X  -165.650, Y  +635.030, Z    +0.000, E1   -48.821, E3 +307947.810}
SPL {X  -165.650, Y  +641.084, Z    +0.000, E1   -48.892, E3 +307958.292}
SPL {X  -165.650, Y  +648.143, Z    +0.000, E1   -49.033, E3 +307969.961}
SPL {X  -165.650, Y  +655.847, Z    +0.000, E1   -48.917, E3 +307984.578}
SPL {X  -165.650, Y  +663.676, Z    +0.000, E1   -48.809, E3 +307999.016}
SPL {X  -165.650, Y  +669.580, Z    +0.000, E1   -48.844, E3 +308009.355}
SPL {X  -165.650, Y  +675.734, Z    +0.000, E1   -49.021, E3 +308019.261}
SPL {X  -165.552, Y  +681.198, Z    +0.000, E1   -48.804, E3 +308030.341}
SPL {X  -165.221, Y  +687.413, Z    +0.000, E1   -48.790, E3 +308041.513}
SPL {X  -164.785, Y  +692.407, Z    +0.000, E1   -48.653, E3 +308051.229}
SPL {X  -164.074, Y  +698.293, Z    +0.000, E1   -48.857, E3 +308060.513}
SPL {X  -163.489, Y  +702.172, Z    +0.000, E1   -48.443, E3 +308069.829}
SPL {X  -162.671, Y  +706.776, Z    +0.000, E1   -48.273, E3 +308079.049}
SPL {X  -161.177, Y  +713.734, Z    +0.000, E1   -48.156, E3 +308092.335}
SPL {X  -159.392, Y  +720.602, Z    +0.000, E1   -47.892, E3 +308105.889}
SPL {X  -157.947, Y  +725.428, Z    +0.000, E1   -47.498, E3 +308116.628}
SPL {X  -156.133, Y  +730.838, Z    +0.000, E1   -47.305, E3 +308127.344}
SPL {X  -153.862, Y  +736.871, Z    +0.000, E1   -47.425, E3 +308137.331}
SPL {X  -143.211, Y  +758.749, Z    +0.000, E1   -53.445, E3 +308140.975}
SPL {X  -130.133, Y  +777.996, Z    +0.000, E1   -46.969, E3 +308236.078}
ENDSPLINE

SPLINE
SPL {X  -153.839, Y  +736.929, Z    +0.000, E1   -32.772, E3 +308309.149}
SPL {X  -162.700, Y  +706.622, Z    +0.000, E1   -19.657, E3 +308313.442}
SPL {X  -164.822, Y  +692.043, Z    +0.000, E1   -12.043, E3 +308309.081}
SPL {X  -165.501, Y  +682.513, Z    +0.000, E1    -6.586, E3 +308307.775}
SPL {X  -165.645, Y  +676.829, Z    +0.000, E1    -2.974, E3 +308307.119}
SPL {X  -165.650, Y  +673.338, Z    +0.000, E1    -0.547, E3 +308306.288}
SPL {X  -165.650, Y  +670.475, Z    +0.000, E1    +1.794, E3 +308306.212}
SPL {X  -165.650, Y  +667.655, Z    +0.000, E1    +4.420, E3 +308306.008}
SPL {X  -165.650, Y  +664.048, Z    +0.000, E1    +8.230, E3 +308305.384}
SPL {X  -165.650, Y  +658.867, Z    +0.000, E1   +14.313, E3 +308303.848}
SPL {X  -165.650, Y  +650.683, Z    +0.000, E1   +24.801, E3 +308301.284}
SPL {X  -165.650, Y  +640.858, Z    +0.000, E1   +34.904, E3 +308303.027}
SPL {X  -165.650, Y  +633.111, Z    +0.000, E1   +43.522, E3 +308299.921}
SPL {X  -165.650, Y  +594.935, Z    +0.000, E1   +58.150, E3 +308314.521}
SPL {X  -165.650, Y  +579.579, Z    +0.000, E1   +60.394, E3 +308322.405}
SPL {X  -165.650, Y  +536.483, Z    +0.000, E1   +57.139, E3 +308380.687}
ENDSPLINE

SPLINE
SPL {X  -165.650, Y  +561.248, Z    +0.000, E1   +49.247, E3 +308391.377}
ENDSPLINE

SPLINE
SPL {X  -165.650, Y  +558.330, Z    +0.000, E1   +47.867, E3 +308405.102}
SPL {X  -165.650, Y  +550.626, Z    +0.000, E1   +48.045, E3 +308418.112}
SPL {X  -165.650, Y  +545.464, Z    +0.000, E1   +47.668, E3 +308429.980}
SPL {X  -165.650, Y  +535.912, Z    +0.000, E1   +47.888, E3 +308446.566}
SPL {X  -165.650, Y  +526.169, Z    +0.000, E1   +47.853, E3 +308464.746}
SPL {X  -165.650, Y  +517.493, Z    +0.000, E1   +47.895, E3 +308480.494}
SPL {X  -165.650, Y  +511.255, Z    +0.000, E1   +47.920, E3 +308491.783}
SPL {X  -165.650, Y  +507.257, Z    +0.000, E1   +47.748, E3 +308500.165}
SPL {X  -165.650, Y  +501.812, Z    +0.000, E1   +47.738, E3 +308510.448}
SPL {X  -165.650, Y  +493.465, Z    +0.000, E1   +47.959, E3 +308524.619}
SPL {X  -165.650, Y  +486.149, Z    +0.000, E1   +47.831, E3 +308538.894}
SPL {X  -165.650, Y  +479.821, Z    +0.000, E1   +47.727, E3 +308551.167}
SPL {X  -165.650, Y  +472.739, Z    +0.000, E1   +47.923, E3 +308563.187}
SPL {X  -165.650, Y  +466.586, Z    +0.000, E1   +48.125, E3 +308573.201}
SPL {X  -165.650, Y  +464.575, Z    +0.000, E1   +47.451, E3 +308580.967}
SPL {X  -165.650, Y  +457.811, Z    +0.000, E1   +47.987, E3 +308590.383}
SPL {X  -165.650, Y  +451.187, Z    +0.000, E1   +47.917, E3 +308603.126}
SPL {X  -165.650, Y  +439.019, Z    +0.000, E1   +49.830, E3 +308613.449}
SPL {X  -165.650, Y  +435.473, Z    +0.000, E1   +49.263, E3 +308623.170}
SPL {X  -165.650, Y  +428.379, Z    +0.000, E1   +49.373, E3 +308634.942}
SPL {X  -165.650, Y  +423.272, Z    +0.000, E1   +49.176, E3 +308645.078}
SPL {X  -165.650, Y  +416.522, Z    +0.000, E1   +49.338, E3 +308656.055}
SPL {X  -165.650, Y  +408.142, Z    +0.000, E1   +49.261, E3 +308671.416}
SPL {X  -165.650, Y  +400.266, Z    +0.000, E1   +49.362, E3 +308684.478}
SPL {X  -165.650, Y  +393.708, Z    +0.000, E1   +49.252, E3 +308696.784}
SPL {X  -165.650, Y  +384.475, Z    +0.000, E1   +49.187, E3 +308713.583}
SPL {X  -165.626, Y  +375.686, Z    +0.000, E1   +49.367, E3 +308727.800}
SPL {X  -165.370, Y  +368.879, Z    +0.000, E1   +49.286, E3 +308740.354}
SPL {X  -164.828, Y  +362.023, Z    +0.000, E1   +48.964, E3 +308754.315}
SPL {X  -164.139, Y  +356.180, Z    +0.000, E1   +49.110, E3 +308763.665}
SPL {X  -163.224, Y  +350.255, Z    +0.000, E1   +48.882, E3 +308775.660}
SPL {X  -162.125, Y  +344.507, Z    +0.000, E1   +48.543, E3 +308787.508}
SPL {X  -160.947, Y  +339.310, Z    +0.000, E1   +48.561, E3 +308796.617}
SPL {X  -159.499, Y  +333.778, Z    +0.000, E1   +48.145, E3 +308808.729}
SPL {X  -157.957, Y  +328.606, Z    +0.000, E1   +47.890, E3 +308819.154}
SPL {X  -156.095, Y  +323.055, Z    +0.000, E1   +47.566, E3 +308830.838}
SPL {X  -153.706, Y  +316.739, Z    +0.000, E1   +47.523, E3 +308841.992}
SPL {X  -143.727, Y  +296.145, Z    +0.000, E1   +53.260, E3 +308845.135}
SPL {X  -128.440, Y  +273.891, Z    +0.000, E1   +47.966, E3 +308932.382}
ENDSPLINE

SPLINE
SPL {X  -131.798, Y  +278.155, Z    +0.000, E1   +45.574, E3 +308958.009}
SPL {X  -154.181, Y  +317.936, Z    +0.000, E1   +32.662, E3 +309023.345}
SPL {X  -162.537, Y  +346.536, Z    +0.000, E1   +20.123, E3 +309022.566}
SPL {X  -164.610, Y  +359.970, Z    +0.000, E1   +13.118, E3 +309017.432}
SPL {X  -165.367, Y  +368.828, Z    +0.000, E1    +8.137, E3 +309015.885}
SPL {X  -165.621, Y  +375.422, Z    +0.000, E1    +4.067, E3 +309016.762}
SPL {X  -165.650, Y  +380.991, Z    +0.000, E1    +0.306, E3 +309014.773}
SPL {X  -165.650, Y  +386.066, Z    +0.000, E1    -4.211, E3 +309014.169}
SPL {X  -165.650, Y  +392.013, Z    +0.000, E1   -10.856, E3 +309013.151}
SPL {X  -165.650, Y  +398.769, Z    +0.000, E1   -19.304, E3 +309011.762}
SPL {X  -165.650, Y  +410.885, Z    +0.000, E1   -34.864, E3 +309007.438}
SPL {X  -165.650, Y  +446.037, Z    +0.000, E1   -53.739, E3 +309021.503}
SPL {X  -165.650, Y  +454.158, Z    +0.000, E1   -53.343, E3 +309031.855}
SPL {X  -165.650, Y  +513.780, Z    +0.000, E1   -56.183, E3 +309092.652}
ENDSPLINE

SPLINE
SPL {X  -165.650, Y  +495.869, Z    +0.000, E1   -48.812, E3 +309108.840}
ENDSPLINE

SPLINE
SPL {X  -165.650, Y  +504.906, Z    +0.000, E1   -48.979, E3 +309124.160}
SPL {X  -165.650, Y  +512.952, Z    +0.000, E1   -48.898, E3 +309138.781}
SPL {X  -165.650, Y  +519.321, Z    +0.000, E1   -49.041, E3 +309149.249}
SPL {X  -165.650, Y  +524.312, Z    +0.000, E1   -48.855, E3 +309159.275}
SPL {X  -165.650, Y  +530.631, Z    +0.000, E1   -48.990, E3 +309169.735}
SPL {X  -165.650, Y  +536.725, Z    +0.000, E1   -48.843, E3 +309181.485}
SPL {X  -165.650, Y  +542.959, Z    +0.000, E1   -48.923, E3 +309192.100}
SPL {X  -165.650, Y  +548.939, Z    +0.000, E1   -48.968, E3 +309202.494}
SPL {X  -165.650, Y  +553.607, Z    +0.000, E1   -48.716, E3 +309212.312}
SPL {X  -165.650, Y  +562.368, Z    +0.000, E1   -49.014, E3 +309226.373}
SPL {X  -165.650, Y  +570.317, Z    +0.000, E1   -48.893, E3 +309241.115}
SPL {X  -165.650, Y  +577.487, Z    +0.000, E1   -49.001, E3 +309253.223}
SPL {X  -165.650, Y  +581.837, Z    +0.000, E1   -48.612, E3 +309263.257}
SPL {X  -165.650, Y  +588.614, Z    +0.000, E1   -49.053, E3 +309272.775}
SPL {X  -165.650, Y  +593.784, Z    +0.000, E1   -48.711, E3 +309284.060}
SPL {X  -165.650, Y  +600.281, Z    +0.000, E1   -48.957, E3 +309294.163}
SPL {X  -165.650, Y  +606.252, Z    +0.000, E1   -48.984, E3 +309304.696}
SPL {X  -165.650, Y  +612.690, Z    +0.000, E1   -49.044, E3 +309315.725}
SPL {X  -165.650, Y  +617.274, Z    +0.000, E1   -48.670, E3 +309326.174}
SPL {X  -165.650, Y  +624.267, Z    +0.000, E1   -48.953, E3 +309336.986}
SPL {X  -165.650, Y  +632.510, Z    +0.000, E1   -48.976, E3 +309351.740}
SPL {X  -165.650, Y  +641.084, Z    +0.000, E1   -48.892, E3 +309367.383}
SPL {X  -165.650, Y  +648.143, Z    +0.000, E1   -49.033, E3 +309379.052}
SPL {X  -165.650, Y  +652.108, Z    +0.000, E1   -48.593, E3 +309388.736}
SPL {X  -165.650, Y  +658.753, Z    +0.000, E1   -49.107, E3 +309397.562}
SPL {X  -165.650, Y  +663.676, Z    +0.000, E1   -48.809, E3 +309408.107}
SPL {X  -165.650, Y  +669.580, Z    +0.000, E1   -48.844, E3 +309418.446}
SPL {X  -165.650, Y  +675.734, Z    +0.000, E1   -49.021, E3 +309428.352}
SPL {X  -165.552, Y  +681.198, Z    +0.000, E1   -48.804, E3 +309439.432}
SPL {X  -165.221, Y  +687.413, Z    +0.000, E1   -48.790, E3 +309450.604}
SPL {X  -164.785, Y  +692.407, Z    +0.000, E1   -48.653, E3 +309460.320}
SPL {X  -164.074, Y  +698.293, Z    +0.000, E1   -48.857, E3 +309469.604}
SPL {X  -163.489, Y  +702.172, Z    +0.000, E1   -48.443, E3 +309478.920}
SPL {X  -162.217, Y  +709.048, Z    +0.000, E1   -48.328, E3 +309492.060}
SPL {X  -160.800, Y  +715.289, Z    +0.000, E1   -47.964, E3 +309505.068}
SPL {X  -159.392, Y  +720.602, Z    +0.000, E1   -47.892, E3 +309514.980}
SPL {X  -157.947, Y  +725.428, Z    +0.000, E1   -47.498, E3 +309525.719}
SPL {X  -156.133, Y  +730.838, Z    +0.000, E1   -47.305, E3 +309536.435}
SPL {X  -153.862, Y  +736.871, Z    +0.000, E1   -47.425, E3 +309546.422}
SPL {X  -143.211, Y  +758.749, Z    +0.000, E1   -53.445, E3 +309550.066}
SPL {X  -129.526, Y  +778.761, Z    +0.000, E1   -47.396, E3 +309640.808}
ENDSPLINE

SPLINE
SPL {X  -152.848, Y  +739.355, Z    +0.000, E1   -33.672, E3 +309716.377}
SPL {X  -162.700, Y  +706.622, Z    +0.000, E1   -19.657, E3 +309722.533}
SPL {X  -164.822, Y  +692.043, Z    +0.000, E1   -12.043, E3 +309718.172}
SPL {X  -165.501, Y  +682.513, Z    +0.000, E1    -6.586, E3 +309716.866}
SPL {X  -165.645, Y  +676.829, Z    +0.000, E1    -2.974, E3 +309716.210}
SPL {X  -165.650, Y  +673.338, Z    +0.000, E1    -0.547, E3 +309715.379}
SPL {X  -165.650, Y  +670.475, Z    +0.000, E1    +1.794, E3 +309715.303}
SPL {X  -165.650, Y  +667.655, Z    +0.000, E1    +4.420, E3 +309715.099}
SPL {X  -165.650, Y  +664.048, Z    +0.000, E1    +8.230, E3 +309714.475}
SPL {X  -165.650, Y  +658.867, Z    +0.000, E1   +14.313, E3 +309712.939}
SPL {X  -165.650, Y  +650.683, Z    +0.000, E1   +24.801, E3 +309710.375}
SPL {X  -165.650, Y  +636.402, Z    +0.000, E1   +39.824, E3 +309710.337}
SPL {X  -165.650, Y  +586.376, Z    +0.000, E1   +59.481, E3 +309728.010}
SPL {X  -165.650, Y  +558.853, Z    +0.000, E1   +50.142, E3 +309799.480}
SPL {X  -165.650, Y  +558.330, Z    +0.000, E1   +47.867, E3 +309814.193}
SPL {X  -165.650, Y  +549.545, Z    +0.000, E1   +47.953, E3 +309829.864}
SPL {X  -165.650, Y  +541.974, Z    +0.000, E1   +47.882, E3 +309844.254}
SPL {X  -165.650, Y  +535.023, Z    +0.000, E1   +47.697, E3 +309858.243}
SPL {X  -165.650, Y  +526.169, Z    +0.000, E1   +47.853, E3 +309873.837}
SPL {X  -165.650, Y  +517.493, Z    +0.000, E1   +47.895, E3 +309889.585}
SPL {X  -165.650, Y  +509.413, Z    +0.000, E1   +47.884, E3 +309904.664}
SPL {X  -165.650, Y  +501.812, Z    +0.000, E1   +47.738, E3 +309919.539}
SPL {X  -165.650, Y  +493.465, Z    +0.000, E1   +47.959, E3 +309933.710}
SPL {X  -165.650, Y  +486.149, Z    +0.000, E1   +47.831, E3 +309947.984}
SPL {X  -165.650, Y  +479.821, Z    +0.000, E1   +47.727, E3 +309960.258}
SPL {X  -165.650, Y  +472.739, Z    +0.000, E1   +47.923, E3 +309972.277}
SPL {X  -165.650, Y  +466.586, Z    +0.000, E1   +48.125, E3 +309982.292}
SPL {X  -165.650, Y  +464.575, Z    +0.000, E1   +47.451, E3 +309990.058}
SPL {X  -165.650, Y  +456.851, Z    +0.000, E1   +47.856, E3 +310002.164}
SPL {X  -165.650, Y  +449.262, Z    +0.000, E1   +48.080, E3 +310014.729}
SPL {X  -165.650, Y  +436.765, Z    +0.000, E1   +49.819, E3 +310026.628}
SPL {X  -165.650, Y  +430.891, Z    +0.000, E1   +49.130, E3 +310041.130}
SPL {X  -165.650, Y  +423.272, Z    +0.000, E1   +49.176, E3 +310054.169}
SPL {X  -165.650, Y  +416.522, Z    +0.000, E1   +49.338, E3 +310065.146}
SPL {X  -165.650, Y  +408.142, Z    +0.000, E1   +49.261, E3 +310080.507}
SPL {X  -165.650, Y  +400.266, Z    +0.000, E1   +49.362, E3 +310093.569}
SPL {X  -165.650, Y  +393.708, Z    +0.000, E1   +49.252, E3 +310105.875}
SPL {X  -165.650, Y  +384.475, Z    +0.000, E1   +49.187, E3 +310122.674}
SPL {X  -165.626, Y  +375.686, Z    +0.000, E1   +49.367, E3 +310136.891}
SPL {X  -165.370, Y  +368.879, Z    +0.000, E1   +49.286, E3 +310149.445}
SPL {X  -164.828, Y  +362.023, Z    +0.000, E1   +48.964, E3 +310163.406}
SPL {X  -164.139, Y  +356.180, Z    +0.000, E1   +49.110, E3 +310172.756}
SPL {X  -163.224, Y  +350.255, Z    +0.000, E1   +48.882, E3 +310184.750}
SPL {X  -162.125, Y  +344.507, Z    +0.000, E1   +48.543, E3 +310196.599}
SPL {X  -160.947, Y  +339.310, Z    +0.000, E1   +48.561, E3 +310205.708}
SPL {X  -159.499, Y  +333.778, Z    +0.000, E1   +48.145, E3 +310217.820}
SPL {X  -157.957, Y  +328.606, Z    +0.000, E1   +47.890, E3 +310228.245}
SPL {X  -156.095, Y  +323.055, Z    +0.000, E1   +47.566, E3 +310239.929}
SPL {X  -153.706, Y  +316.739, Z    +0.000, E1   +47.523, E3 +310251.083}
SPL {X  -143.727, Y  +296.145, Z    +0.000, E1   +53.260, E3 +310254.226}
SPL {X  -128.440, Y  +273.891, Z    +0.000, E1   +47.966, E3 +310341.473}
ENDSPLINE

SPLINE
SPL {X  -131.798, Y  +278.155, Z    +0.000, E1   +45.574, E3 +310367.100}
SPL {X  -154.181, Y  +317.936, Z    +0.000, E1   +32.662, E3 +310432.436}
SPL {X  -162.537, Y  +346.536, Z    +0.000, E1   +20.123, E3 +310431.657}
SPL {X  -165.197, Y  +366.255, Z    +0.000, E1    +9.700, E3 +310425.452}
SPL {X  -165.621, Y  +375.422, Z    +0.000, E1    +4.067, E3 +310425.853}
SPL {X  -165.650, Y  +379.733, Z    +0.000, E1    +1.160, E3 +310424.159}
SPL {X  -165.650, Y  +383.552, Z    +0.000, E1    -1.868, E3 +310423.408}
SPL {X  -165.650, Y  +387.323, Z    +0.000, E1    -5.609, E3 +310423.225}
SPL {X  -165.650, Y  +392.013, Z    +0.000, E1   -10.856, E3 +310422.242}
SPL {X  -165.650, Y  +398.769, Z    +0.000, E1   -19.304, E3 +310420.853}
SPL {X  -165.650, Y  +410.885, Z    +0.000, E1   -34.864, E3 +310416.529}
SPL {X  -165.650, Y  +446.037, Z    +0.000, E1   -53.739, E3 +310430.594}
SPL {X  -165.650, Y  +454.158, Z    +0.000, E1   -53.343, E3 +310440.945}
SPL {X  -165.650, Y  +513.780, Z    +0.000, E1   -56.183, E3 +310501.742}
ENDSPLINE

SPLINE
SPL {X  -165.650, Y  +495.869, Z    +0.000, E1   -48.812, E3 +310517.931}
ENDSPLINE

SPLINE
SPL {X  -165.650, Y  +504.906, Z    +0.000, E1   -48.979, E3 +310533.251}
SPL {X  -165.650, Y  +512.952, Z    +0.000, E1   -48.898, E3 +310547.872}
SPL {X  -165.650, Y  +519.321, Z    +0.000, E1   -49.041, E3 +310558.340}
SPL {X  -165.650, Y  +524.312, Z    +0.000, E1   -48.855, E3 +310568.366}
SPL {X  -165.650, Y  +530.631, Z    +0.000, E1   -48.990, E3 +310578.826}
SPL {X  -165.650, Y  +536.725, Z    +0.000, E1   -48.843, E3 +310590.576}
SPL {X  -165.650, Y  +542.959, Z    +0.000, E1   -48.923, E3 +310601.191}
SPL {X  -165.650, Y  +548.939, Z    +0.000, E1   -48.968, E3 +310611.585}
SPL {X  -165.650, Y  +553.607, Z    +0.000, E1   -48.716, E3 +310621.403}
SPL {X  -165.650, Y  +562.368, Z    +0.000, E1   -49.014, E3 +310635.464}
SPL {X  -165.650, Y  +570.317, Z    +0.000, E1   -48.893, E3 +310650.206}
SPL {X  -165.650, Y  +577.487, Z    +0.000, E1   -49.001, E3 +310662.314}
SPL {X  -165.650, Y  +581.837, Z    +0.000, E1   -48.612, E3 +310672.348}
SPL {X  -165.650, Y  +588.614, Z    +0.000, E1   -49.053, E3 +310681.865}
SPL {X  -165.650, Y  +593.784, Z    +0.000, E1   -48.711, E3 +310693.151}
SPL {X  -165.650, Y  +600.281, Z    +0.000, E1   -48.957, E3 +310703.253}
SPL {X  -165.650, Y  +606.252, Z    +0.000, E1   -48.984, E3 +310713.787}
SPL {X  -165.650, Y  +612.690, Z    +0.000, E1   -49.044, E3 +310724.816}
SPL {X  -165.650, Y  +617.274, Z    +0.000, E1   -48.670, E3 +310735.265}
SPL {X  -165.650, Y  +624.267, Z    +0.000, E1   -48.953, E3 +310746.076}
SPL {X  -165.650, Y  +632.510, Z    +0.000, E1   -48.976, E3 +310760.831}
SPL {X  -165.650, Y  +641.084, Z    +0.000, E1   -48.892, E3 +310776.474}
SPL {X  -165.650, Y  +648.143, Z    +0.000, E1   -49.033, E3 +310788.143}
SPL {X  -165.650, Y  +655.847, Z    +0.000, E1   -48.917, E3 +310802.760}
SPL {X  -165.650, Y  +663.676, Z    +0.000, E1   -48.809, E3 +310817.198}
SPL {X  -165.650, Y  +669.580, Z    +0.000, E1   -48.844, E3 +310827.537}
SPL {X  -165.650, Y  +675.734, Z    +0.000, E1   -49.021, E3 +310837.443}
SPL {X  -165.552, Y  +681.198, Z    +0.000, E1   -48.804, E3 +310848.523}
SPL {X  -165.221, Y  +687.413, Z    +0.000, E1   -48.790, E3 +310859.695}
SPL {X  -164.785, Y  +692.407, Z    +0.000, E1   -48.653, E3 +310869.410}
SPL {X  -164.074, Y  +698.293, Z    +0.000, E1   -48.857, E3 +310878.695}
SPL {X  -163.489, Y  +702.172, Z    +0.000, E1   -48.443, E3 +310888.011}
SPL {X  -162.671, Y  +706.776, Z    +0.000, E1   -48.273, E3 +310897.230}
SPL {X  -161.177, Y  +713.734, Z    +0.000, E1   -48.156, E3 +310910.517}
SPL {X  -159.392, Y  +720.602, Z    +0.000, E1   -47.892, E3 +310924.070}
SPL {X  -157.947, Y  +725.428, Z    +0.000, E1   -47.498, E3 +310934.810}
SPL {X  -155.696, Y  +732.057, Z    +0.000, E1   -47.224, E3 +310948.286}
SPL {X  -152.475, Y  +740.240, Z    +0.000, E1   -48.059, E3 +310958.116}
SPL {X  -143.211, Y  +758.749, Z    +0.000, E1   -53.445, E3 +310959.157}
SPL {X  -129.526, Y  +778.761, Z    +0.000, E1   -47.396, E3 +311049.898}
ENDSPLINE

SPLINE
SPL {X  -152.848, Y  +739.355, Z    +0.000, E1   -33.672, E3 +311125.467}
SPL {X  -162.700, Y  +706.622, Z    +0.000, E1   -19.657, E3 +311131.624}
SPL {X  -164.822, Y  +692.043, Z    +0.000, E1   -12.043, E3 +311127.263}
SPL {X  -165.501, Y  +682.513, Z    +0.000, E1    -6.586, E3 +311125.957}
SPL {X  -165.650, Y  +674.436, Z    +0.000, E1    -1.443, E3 +311124.732}
SPL {X  -165.650, Y  +669.008, Z    +0.000, E1    +2.993, E3 +311124.287}
SPL {X  -165.650, Y  +663.208, Z    +0.000, E1    +9.118, E3 +311123.372}
SPL {X  -165.650, Y  +657.399, Z    +0.000, E1   +16.251, E3 +311121.491}
SPL {X  -165.650, Y  +650.683, Z    +0.000, E1   +24.801, E3 +311119.466}
SPL {X  -165.650, Y  +636.402, Z    +0.000, E1   +39.824, E3 +311119.428}
SPL {X  -165.650, Y  +594.935, Z    +0.000, E1   +58.150, E3 +311132.703}
SPL {X  -165.650, Y  +579.579, Z    +0.000, E1   +60.394, E3 +311140.587}
SPL {X  -165.650, Y  +554.310, Z    +0.000, E1   +51.914, E3 +311205.145}
ENDSPLINE

SPLINE
SPL {X  -165.650, Y  +561.648, Z    +0.000, E1   +48.058, E3 +311215.962}
ENDSPLINE

SPLINE
SPL {X  -165.650, Y  +556.469, Z    +0.000, E1   +47.823, E3 +311226.830}
SPL {X  -165.650, Y  +550.626, Z    +0.000, E1   +48.045, E3 +311236.294}
SPL {X  -165.650, Y  +545.464, Z    +0.000, E1   +47.668, E3 +311248.162}
SPL {X  -165.650, Y  +537.837, Z    +0.000, E1   +47.880, E3 +311261.040}
SPL {X  -165.650, Y  +530.616, Z    +0.000, E1   +47.886, E3 +311274.405}
SPL {X  -165.650, Y  +524.679, Z    +0.000, E1   +47.721, E3 +311286.297}
SPL {X  -165.650, Y  +517.493, Z    +0.000, E1   +47.895, E3 +311298.676}
SPL {X  -165.650, Y  +511.255, Z    +0.000, E1   +47.920, E3 +311309.965}
SPL {X  -165.650, Y  +507.257, Z    +0.000, E1   +47.748, E3 +311318.347}
SPL {X  -165.650, Y  +501.812, Z    +0.000, E1   +47.738, E3 +311328.630}
SPL {X  -165.650, Y  +493.465, Z    +0.000, E1   +47.959, E3 +311342.800}
SPL {X  -165.650, Y  +486.149, Z    +0.000, E1   +47.831, E3 +311357.075}
SPL {X  -165.650, Y  +477.718, Z    +0.000, E1   +47.870, E3 +311372.515}
SPL {X  -165.650, Y  +469.088, Z    +0.000, E1   +47.982, E3 +311387.734}
SPL {X  -165.650, Y  +464.575, Z    +0.000, E1   +47.451, E3 +311399.149}
SPL {X  -165.650, Y  +456.851, Z    +0.000, E1   +47.856, E3 +311411.254}
SPL {X  -165.650, Y  +449.262, Z    +0.000, E1   +48.080, E3 +311423.820}
SPL {X  -165.650, Y  +436.454, Z    +0.000, E1   +49.483, E3 +311438.527}
SPL {X  -165.650, Y  +428.379, Z    +0.000, E1   +49.373, E3 +311453.124}
SPL {X  -165.650, Y  +423.272, Z    +0.000, E1   +49.176, E3 +311463.259}
SPL {X  -165.650, Y  +416.522, Z    +0.000, E1   +49.338, E3 +311474.237}
SPL {X  -165.650, Y  +410.777, Z    +0.000, E1   +49.173, E3 +311485.290}
SPL {X  -165.650, Y  +405.230, Z    +0.000, E1   +49.266, E3 +311494.493}
SPL {X  -165.650, Y  +398.850, Z    +0.000, E1   +49.279, E3 +311505.784}
SPL {X  -165.650, Y  +391.803, Z    +0.000, E1   +49.319, E3 +311517.822}
SPL {X  -165.650, Y  +384.475, Z    +0.000, E1   +49.187, E3 +311531.765}
SPL {X  -165.602, Y  +374.507, Z    +0.000, E1   +49.269, E3 +311548.788}
SPL {X  -165.255, Y  +367.073, Z    +0.000, E1   +49.394, E3 +311560.981}
SPL {X  -164.828, Y  +362.023, Z    +0.000, E1   +48.964, E3 +311572.497}
SPL {X  -163.908, Y  +354.543, Z    +0.000, E1   +49.169, E3 +311584.444}
SPL {X  -163.052, Y  +349.277, Z    +0.000, E1   +48.680, E3 +311596.550}
SPL {X  -162.125, Y  +344.507, Z    +0.000, E1   +48.543, E3 +311605.690}
SPL {X  -160.947, Y  +339.310, Z    +0.000, E1   +48.561, E3 +311614.799}
SPL {X  -159.860, Y  +335.086, Z    +0.000, E1   +48.145, E3 +311624.511}
SPL {X  -158.277, Y  +329.631, Z    +0.000, E1   +47.981, E3 +311635.133}
SPL {X  -156.804, Y  +325.092, Z    +0.000, E1   +47.609, E3 +311645.026}
SPL {X  -155.465, Y  +321.311, Z    +0.000, E1   +47.446, E3 +311652.561}
SPL {X  -153.706, Y  +316.739, Z    +0.000, E1   +47.523, E3 +311660.174}
SPL {X  -143.727, Y  +296.145, Z    +0.000, E1   +53.260, E3 +311663.317}
SPL {X  -128.440, Y  +273.891, Z    +0.000, E1   +47.966, E3 +311750.564}
ENDSPLINE

SPLINE
SPL {X  -131.798, Y  +278.155, Z    +0.000, E1   +45.574, E3 +311776.191}
SPL {X  -154.181, Y  +317.936, Z    +0.000, E1   +32.662, E3 +311841.527}
SPL {X  -162.537, Y  +346.536, Z    +0.000, E1   +20.123, E3 +311840.748}
SPL {X  -164.610, Y  +359.970, Z    +0.000, E1   +13.118, E3 +311835.614}
SPL {X  -165.367, Y  +368.828, Z    +0.000, E1    +8.137, E3 +311834.067}
SPL {X  -165.621, Y  +375.422, Z    +0.000, E1    +4.067, E3 +311834.943}
SPL {X  -165.650, Y  +379.733, Z    +0.000, E1    +1.160, E3 +311833.249}
SPL {X  -165.650, Y  +383.552, Z    +0.000, E1    -1.868, E3 +311832.499}
SPL {X  -165.650, Y  +387.323, Z    +0.000, E1    -5.609, E3 +311832.315}
SPL {X  -165.650, Y  +392.013, Z    +0.000, E1   -10.856, E3 +311831.333}
SPL {X  -165.650, Y  +398.769, Z    +0.000, E1   -19.304, E3 +311829.944}
SPL {X  -165.650, Y  +407.471, Z    +0.000, E1   -31.017, E3 +311826.103}
SPL {X  -165.650, Y  +414.706, Z    +0.000, E1   -39.242, E3 +311825.079}
SPL {X  -165.650, Y  +446.037, Z    +0.000, E1   -53.739, E3 +311839.685}
SPL {X  -165.650, Y  +454.158, Z    +0.000, E1   -53.343, E3 +311850.036}
SPL {X  -165.650, Y  +513.780, Z    +0.000, E1   -56.183, E3 +311910.833}
ENDSPLINE

SPLINE
SPL {X  -165.650, Y  +495.869, Z    +0.000, E1   -48.812, E3 +311927.022}
ENDSPLINE

SPLINE
SPL {X  -165.650, Y  +502.040, Z    +0.000, E1   -48.856, E3 +311937.766}
SPL {X  -165.650, Y  +507.863, Z    +0.000, E1   -49.013, E3 +311947.186}
SPL {X  -165.650, Y  +512.952, Z    +0.000, E1   -48.898, E3 +311956.963}
SPL {X  -165.650, Y  +519.321, Z    +0.000, E1   -49.041, E3 +311967.431}
SPL {X  -165.650, Y  +524.312, Z    +0.000, E1   -48.855, E3 +311977.457}
SPL {X  -165.650, Y  +530.631, Z    +0.000, E1   -48.990, E3 +311987.917}
SPL {X  -165.650, Y  +536.725, Z    +0.000, E1   -48.843, E3 +311999.667}
SPL {X  -165.650, Y  +542.959, Z    +0.000, E1   -48.923, E3 +312010.282}
SPL {X  -165.650, Y  +548.939, Z    +0.000, E1   -48.968, E3 +312020.676}
SPL {X  -165.650, Y  +553.607, Z    +0.000, E1   -48.716, E3 +312030.494}
SPL {X  -165.650, Y  +562.368, Z    +0.000, E1   -49.014, E3 +312044.555}
SPL {X  -165.650, Y  +570.317, Z    +0.000, E1   -48.893, E3 +312059.297}
SPL {X  -165.650, Y  +577.487, Z    +0.000, E1   -49.001, E3 +312071.405}
SPL {X  -165.650, Y  +581.837, Z    +0.000, E1   -48.612, E3 +312081.439}
SPL {X  -165.650, Y  +588.614, Z    +0.000, E1   -49.053, E3 +312090.956}
SPL {X  -165.650, Y  +593.784, Z    +0.000, E1   -48.711, E3 +312102.242}
SPL {X  -165.650, Y  +600.281, Z    +0.000, E1   -48.957, E3 +312112.344}
SPL {X  -165.650, Y  +606.252, Z    +0.000, E1   -48.984, E3 +312122.878}
SPL {X  -165.650, Y  +612.690, Z    +0.000, E1   -49.044, E3 +312133.907}
SPL {X  -165.650, Y  +617.274, Z    +0.000, E1   -48.670, E3 +312144.356}
SPL {X  -165.650, Y  +624.267, Z    +0.000, E1   -48.953, E3 +312155.167}
SPL {X  -165.650, Y  +632.510, Z    +0.000, E1   -48.976, E3 +312169.922}
SPL {X  -165.650, Y  +641.084, Z    +0.000, E1   -48.892, E3 +312185.564}
SPL {X  -165.650, Y  +648.143, Z    +0.000, E1   -49.033, E3 +312197.234}
SPL {X  -165.650, Y  +655.847, Z    +0.000, E1   -48.917, E3 +312211.851}
SPL {X  -165.650, Y  +663.676, Z    +0.000, E1   -48.809, E3 +312226.289}
SPL {X  -165.650, Y  +669.580, Z    +0.000, E1   -48.844, E3 +312236.628}
SPL {X  -165.650, Y  +675.734, Z    +0.000, E1   -49.021, E3 +312246.534}
SPL {X  -165.552, Y  +681.198, Z    +0.000, E1   -48.804, E3 +312257.614}
SPL {X  -165.221, Y  +687.413, Z    +0.000, E1   -48.790, E3 +312268.786}
SPL {X  -164.785, Y  +692.407, Z    +0.000, E1   -48.653, E3 +312278.501}
SPL {X  -164.074, Y  +698.293, Z    +0.000, E1   -48.857, E3 +312287.785}
SPL {X  -163.489, Y  +702.172, Z    +0.000, E1   -48.443, E3 +312297.102}
SPL {X  -162.671, Y  +706.776, Z    +0.000, E1   -48.273, E3 +312306.321}
SPL {X  -161.177, Y  +713.734, Z    +0.000, E1   -48.156, E3 +312319.608}
SPL {X  -159.392, Y  +720.602, Z    +0.000, E1   -47.892, E3 +312333.161}
SPL {X  -157.947, Y  +725.428, Z    +0.000, E1   -47.498, E3 +312343.900}
SPL {X  -155.696, Y  +732.057, Z    +0.000, E1   -47.224, E3 +312357.377}
SPL {X  -152.475, Y  +740.240, Z    +0.000, E1   -48.059, E3 +312367.206}
SPL {X  -143.211, Y  +758.749, Z    +0.000, E1   -53.445, E3 +312368.248}
SPL {X  -129.526, Y  +778.761, Z    +0.000, E1   -47.396, E3 +312458.989}
ENDSPLINE

SPLINE
SPL {X  -152.848, Y  +739.355, Z    +0.000, E1   -33.672, E3 +312534.558}
SPL {X  -162.700, Y  +706.622, Z    +0.000, E1   -19.657, E3 +312540.715}
SPL {X  -164.822, Y  +692.043, Z    +0.000, E1   -12.043, E3 +312536.354}
SPL {X  -165.501, Y  +682.513, Z    +0.000, E1    -6.586, E3 +312535.048}
SPL {X  -165.650, Y  +674.436, Z    +0.000, E1    -1.443, E3 +312533.823}
SPL {X  -165.650, Y  +669.008, Z    +0.000, E1    +2.993, E3 +312533.378}
SPL {X  -165.650, Y  +663.208, Z    +0.000, E1    +9.118, E3 +312532.462}
SPL {X  -165.650, Y  +657.399, Z    +0.000, E1   +16.251, E3 +312530.582}
SPL {X  -165.650, Y  +650.683, Z    +0.000, E1   +24.801, E3 +312528.557}
SPL {X  -165.650, Y  +636.402, Z    +0.000, E1   +39.824, E3 +312528.519}
SPL {X  -165.650, Y  +594.935, Z    +0.000, E1   +58.150, E3 +312541.794}
SPL {X  -165.650, Y  +579.579, Z    +0.000, E1   +60.394, E3 +312549.678}
SPL {X  -165.650, Y  +554.310, Z    +0.000, E1   +51.914, E3 +312614.236}
ENDSPLINE

SPLINE
SPL {X  -165.650, Y  +561.648, Z    +0.000, E1   +48.058, E3 +312625.053}
ENDSPLINE

SPLINE
SPL {X  -165.650, Y  +556.469, Z    +0.000, E1   +47.823, E3 +312635.921}
SPL {X  -165.650, Y  +550.626, Z    +0.000, E1   +48.045, E3 +312645.385}
SPL {X  -165.650, Y  +545.464, Z    +0.000, E1   +47.668, E3 +312657.253}
SPL {X  -165.650, Y  +537.837, Z    +0.000, E1   +47.880, E3 +312670.130}
SPL {X  -165.650, Y  +530.616, Z    +0.000, E1   +47.886, E3 +312683.496}
SPL {X  -165.650, Y  +524.679, Z    +0.000, E1   +47.721, E3 +312695.388}
SPL {X  -165.650, Y  +517.493, Z    +0.000, E1   +47.895, E3 +312707.767}
SPL {X  -165.650, Y  +511.255, Z    +0.000, E1   +47.920, E3 +312719.056}
SPL {X  -165.650, Y  +507.257, Z    +0.000, E1   +47.748, E3 +312727.437}
SPL {X  -165.650, Y  +501.812, Z    +0.000, E1   +47.738, E3 +312737.721}
SPL {X  -165.650, Y  +493.465, Z    +0.000, E1   +47.959, E3 +312751.891}
SPL {X  -165.650, Y  +486.149, Z    +0.000, E1   +47.831, E3 +312766.166}
SPL {X  -165.650, Y  +477.718, Z    +0.000, E1   +47.870, E3 +312781.606}
SPL {X  -165.650, Y  +469.088, Z    +0.000, E1   +47.982, E3 +312796.825}
SPL {X  -165.650, Y  +464.575, Z    +0.000, E1   +47.451, E3 +312808.240}
SPL {X  -165.650, Y  +456.851, Z    +0.000, E1   +47.856, E3 +312820.345}
SPL {X  -165.650, Y  +449.262, Z    +0.000, E1   +48.080, E3 +312832.911}
SPL {X  -165.650, Y  +436.454, Z    +0.000, E1   +49.483, E3 +312847.618}
SPL {X  -165.650, Y  +428.379, Z    +0.000, E1   +49.373, E3 +312862.214}
SPL {X  -165.650, Y  +423.272, Z    +0.000, E1   +49.176, E3 +312872.350}
SPL {X  -165.650, Y  +416.522, Z    +0.000, E1   +49.338, E3 +312883.328}
SPL {X  -165.650, Y  +410.777, Z    +0.000, E1   +49.173, E3 +312894.381}
SPL {X  -165.650, Y  +405.230, Z    +0.000, E1   +49.266, E3 +312903.584}
SPL {X  -165.650, Y  +398.850, Z    +0.000, E1   +49.279, E3 +312914.875}
SPL {X  -165.650, Y  +391.803, Z    +0.000, E1   +49.319, E3 +312926.913}
SPL {X  -165.650, Y  +384.475, Z    +0.000, E1   +49.187, E3 +312940.855}
SPL {X  -165.602, Y  +374.507, Z    +0.000, E1   +49.269, E3 +312957.879}
SPL {X  -165.255, Y  +367.073, Z    +0.000, E1   +49.394, E3 +312970.072}
SPL {X  -164.828, Y  +362.023, Z    +0.000, E1   +48.964, E3 +312981.588}
SPL {X  -163.908, Y  +354.543, Z    +0.000, E1   +49.169, E3 +312993.535}
SPL {X  -163.052, Y  +349.277, Z    +0.000, E1   +48.680, E3 +313005.641}
SPL {X  -162.125, Y  +344.507, Z    +0.000, E1   +48.543, E3 +313014.781}
SPL {X  -160.947, Y  +339.310, Z    +0.000, E1   +48.561, E3 +313023.889}
SPL {X  -159.860, Y  +335.086, Z    +0.000, E1   +48.145, E3 +313033.602}
SPL {X  -158.277, Y  +329.631, Z    +0.000, E1   +47.981, E3 +313044.224}
SPL {X  -156.804, Y  +325.092, Z    +0.000, E1   +47.609, E3 +313054.117}
SPL {X  -155.465, Y  +321.311, Z    +0.000, E1   +47.446, E3 +313061.651}
SPL {X  -153.706, Y  +316.739, Z    +0.000, E1   +47.523, E3 +313069.265}
SPL {X  -143.727, Y  +296.145, Z    +0.000, E1   +53.260, E3 +313072.408}
SPL {X  -128.440, Y  +273.891, Z    +0.000, E1   +47.966, E3 +313159.655}
ENDSPLINE

SPLINE
SPL {X  -131.798, Y  +278.155, Z    +0.000, E1   +45.574, E3 +313185.282}
SPL {X  -154.181, Y  +317.936, Z    +0.000, E1   +32.662, E3 +313250.618}
SPL {X  -162.537, Y  +346.536, Z    +0.000, E1   +20.123, E3 +313249.838}
SPL {X  -164.610, Y  +359.970, Z    +0.000, E1   +13.118, E3 +313244.705}
SPL {X  -165.367, Y  +368.828, Z    +0.000, E1    +8.137, E3 +313243.158}
SPL {X  -165.621, Y  +375.422, Z    +0.000, E1    +4.067, E3 +313244.034}
SPL {X  -165.650, Y  +380.991, Z    +0.000, E1    +0.306, E3 +313242.046}
SPL {X  -165.650, Y  +386.066, Z    +0.000, E1    -4.211, E3 +313241.442}
SPL {X  -165.650, Y  +392.013, Z    +0.000, E1   -10.856, E3 +313240.424}
SPL {X  -165.650, Y  +398.769, Z    +0.000, E1   -19.304, E3 +313239.035}
SPL {X  -165.650, Y  +410.885, Z    +0.000, E1   -34.864, E3 +313234.711}
SPL {X  -165.650, Y  +446.037, Z    +0.000, E1   -53.739, E3 +313248.775}
SPL {X  -165.650, Y  +454.158, Z    +0.000, E1   -53.343, E3 +313259.127}
SPL {X  -165.650, Y  +513.780, Z    +0.000, E1   -56.183, E3 +313319.924}
ENDSPLINE

SPLINE
SPL {X  -165.650, Y  +495.869, Z    +0.000, E1   -48.812, E3 +313336.113}
ENDSPLINE

SPLINE
SPL {X  -165.650, Y  +502.040, Z    +0.000, E1   -48.856, E3 +313346.857}
SPL {X  -165.650, Y  +507.863, Z    +0.000, E1   -49.013, E3 +313356.277}
SPL {X  -165.650, Y  +512.952, Z    +0.000, E1   -48.898, E3 +313366.054}
SPL {X  -165.650, Y  +519.321, Z    +0.000, E1   -49.041, E3 +313376.522}
SPL {X  -165.650, Y  +524.312, Z    +0.000, E1   -48.855, E3 +313386.548}
SPL {X  -165.650, Y  +530.631, Z    +0.000, E1   -48.990, E3 +313397.007}
SPL {X  -165.650, Y  +536.725, Z    +0.000, E1   -48.843, E3 +313408.758}
SPL {X  -165.650, Y  +542.959, Z    +0.000, E1   -48.923, E3 +313419.373}
SPL {X  -165.650, Y  +548.939, Z    +0.000, E1   -48.968, E3 +313429.767}
SPL {X  -165.650, Y  +553.607, Z    +0.000, E1   -48.716, E3 +313439.585}
SPL {X  -165.650, Y  +562.368, Z    +0.000, E1   -49.014, E3 +313453.645}
SPL {X  -165.650, Y  +570.317, Z    +0.000, E1   -48.893, E3 +313468.388}
SPL {X  -165.650, Y  +577.487, Z    +0.000, E1   -49.001, E3 +313480.496}
SPL {X  -165.650, Y  +581.837, Z    +0.000, E1   -48.612, E3 +313490.530}
SPL {X  -165.650, Y  +588.614, Z    +0.000, E1   -49.053, E3 +313500.047}
SPL {X  -165.650, Y  +593.784, Z    +0.000, E1   -48.711, E3 +313511.333}
SPL {X  -165.650, Y  +600.281, Z    +0.000, E1   -48.957, E3 +313521.435}
SPL {X  -165.650, Y  +606.252, Z    +0.000, E1   -48.984, E3 +313531.969}
SPL {X  -165.650, Y  +612.690, Z    +0.000, E1   -49.044, E3 +313542.997}
SPL {X  -165.650, Y  +617.274, Z    +0.000, E1   -48.670, E3 +313553.447}
SPL {X  -165.650, Y  +624.267, Z    +0.000, E1   -48.953, E3 +313564.258}
SPL {X  -165.650, Y  +632.510, Z    +0.000, E1   -48.976, E3 +313579.013}
SPL {X  -165.650, Y  +641.084, Z    +0.000, E1   -48.892, E3 +313594.655}
SPL {X  -165.650, Y  +648.143, Z    +0.000, E1   -49.033, E3 +313606.324}
SPL {X  -165.650, Y  +655.847, Z    +0.000, E1   -48.917, E3 +313620.942}
SPL {X  -165.650, Y  +663.676, Z    +0.000, E1   -48.809, E3 +313635.380}
SPL {X  -165.650, Y  +669.580, Z    +0.000, E1   -48.844, E3 +313645.719}
SPL {X  -165.650, Y  +675.734, Z    +0.000, E1   -49.021, E3 +313655.625}
SPL {X  -165.552, Y  +681.198, Z    +0.000, E1   -48.804, E3 +313666.705}
SPL {X  -165.221, Y  +687.413, Z    +0.000, E1   -48.790, E3 +313677.877}
SPL {X  -164.785, Y  +692.407, Z    +0.000, E1   -48.653, E3 +313687.592}
SPL {X  -164.074, Y  +698.293, Z    +0.000, E1   -48.857, E3 +313696.876}
SPL {X  -163.489, Y  +702.172, Z    +0.000, E1   -48.443, E3 +313706.193}
SPL {X  -162.217, Y  +709.048, Z    +0.000, E1   -48.328, E3 +313719.333}
SPL {X  -160.800, Y  +715.289, Z    +0.000, E1   -47.964, E3 +313732.341}
SPL {X  -159.392, Y  +720.602, Z    +0.000, E1   -47.892, E3 +313742.252}
SPL {X  -157.947, Y  +725.428, Z    +0.000, E1   -47.498, E3 +313752.991}
SPL {X  -155.696, Y  +732.057, Z    +0.000, E1   -47.224, E3 +313766.468}
SPL {X  -152.475, Y  +740.240, Z    +0.000, E1   -48.059, E3 +313776.297}
SPL {X  -143.211, Y  +758.749, Z    +0.000, E1   -53.445, E3 +313777.339}
SPL {X  -129.526, Y  +778.761, Z    +0.000, E1   -47.396, E3 +313868.080}
ENDSPLINE

SPLINE
SPL {X  -152.848, Y  +739.355, Z    +0.000, E1   -33.672, E3 +313943.649}
SPL {X  -162.700, Y  +706.622, Z    +0.000, E1   -19.657, E3 +313949.806}
SPL {X  -164.822, Y  +692.043, Z    +0.000, E1   -12.043, E3 +313945.445}
SPL {X  -165.501, Y  +682.513, Z    +0.000, E1    -6.586, E3 +313944.139}
SPL {X  -165.650, Y  +674.436, Z    +0.000, E1    -1.443, E3 +313942.914}
SPL {X  -165.650, Y  +670.475, Z    +0.000, E1    +1.794, E3 +313942.575}
SPL {X  -165.650, Y  +667.655, Z    +0.000, E1    +4.420, E3 +313942.371}
SPL {X  -165.650, Y  +663.208, Z    +0.000, E1    +9.118, E3 +313941.553}
SPL {X  -165.650, Y  +657.399, Z    +0.000, E1   +16.251, E3 +313939.673}
SPL {X  -165.650, Y  +650.683, Z    +0.000, E1   +24.801, E3 +313937.647}
SPL {X  -165.650, Y  +636.402, Z    +0.000, E1   +39.824, E3 +313937.610}
SPL {X  -165.650, Y  +586.376, Z    +0.000, E1   +59.481, E3 +313955.283}
SPL {X  -165.650, Y  +554.310, Z    +0.000, E1   +51.914, E3 +314023.327}
ENDSPLINE

SPLINE
SPL {X  -165.650, Y  +561.648, Z    +0.000, E1   +48.058, E3 +314034.144}
ENDSPLINE

SPLINE
SPL {X  -165.650, Y  +556.469, Z    +0.000, E1   +47.823, E3 +314045.012}
SPL {X  -165.650, Y  +549.545, Z    +0.000, E1   +47.953, E3 +314057.137}
SPL {X  -165.650, Y  +541.974, Z    +0.000, E1   +47.882, E3 +314071.527}
SPL {X  -165.650, Y  +535.023, Z    +0.000, E1   +47.697, E3 +314085.515}
SPL {X  -165.650, Y  +526.169, Z    +0.000, E1   +47.853, E3 +314101.110}
SPL {X  -165.650, Y  +517.493, Z    +0.000, E1   +47.895, E3 +314116.858}
SPL {X  -165.650, Y  +509.413, Z    +0.000, E1   +47.884, E3 +314131.937}
SPL {X  -165.650, Y  +501.812, Z    +0.000, E1   +47.738, E3 +314146.812}
SPL {X  -165.650, Y  +494.522, Z    +0.000, E1   +48.055, E3 +314158.339}
SPL {X  -165.650, Y  +489.529, Z    +0.000, E1   +47.849, E3 +314168.792}
SPL {X  -165.650, Y  +481.894, Z    +0.000, E1   +47.756, E3 +314183.693}
SPL {X  -165.650, Y  +472.739, Z    +0.000, E1   +47.923, E3 +314199.550}
SPL {X  -165.650, Y  +466.586, Z    +0.000, E1   +48.125, E3 +314209.565}
SPL {X  -165.650, Y  +464.575, Z    +0.000, E1   +47.451, E3 +314217.330}
SPL {X  -165.650, Y  +457.811, Z    +0.000, E1   +47.987, E3 +314226.747}
SPL {X  -165.650, Y  +451.187, Z    +0.000, E1   +47.917, E3 +314239.490}
SPL {X  -165.650, Y  +436.454, Z    +0.000, E1   +49.483, E3 +314256.709}
SPL {X  -165.650, Y  +428.379, Z    +0.000, E1   +49.373, E3 +314271.305}
SPL {X  -165.650, Y  +423.272, Z    +0.000, E1   +49.176, E3 +314281.441}
SPL {X  -165.650, Y  +416.522, Z    +0.000, E1   +49.338, E3 +314292.419}
SPL {X  -165.650, Y  +408.142, Z    +0.000, E1   +49.261, E3 +314307.780}
SPL {X  -165.650, Y  +400.266, Z    +0.000, E1   +49.362, E3 +314320.841}
SPL {X  -165.650, Y  +393.708, Z    +0.000, E1   +49.252, E3 +314333.148}
SPL {X  -165.650, Y  +384.475, Z    +0.000, E1   +49.187, E3 +314349.946}
SPL {X  -165.602, Y  +374.507, Z    +0.000, E1   +49.269, E3 +314366.970}
SPL {X  -165.183, Y  +366.070, Z    +0.000, E1   +49.261, E3 +314381.854}
SPL {X  -164.692, Y  +360.715, Z    +0.000, E1   +48.960, E3 +314392.935}
SPL {X  -163.908, Y  +354.543, Z    +0.000, E1   +49.169, E3 +314402.626}
SPL {X  -163.052, Y  +349.277, Z    +0.000, E1   +48.680, E3 +314414.732}
SPL {X  -162.125, Y  +344.507, Z    +0.000, E1   +48.543, E3 +314423.871}
SPL {X  -160.947, Y  +339.310, Z    +0.000, E1   +48.561, E3 +314432.980}
SPL {X  -159.499, Y  +333.778, Z    +0.000, E1   +48.145, E3 +314445.093}
SPL {X  -157.957, Y  +328.606, Z    +0.000, E1   +47.890, E3 +314455.517}
SPL {X  -156.095, Y  +323.055, Z    +0.000, E1   +47.566, E3 +314467.202}
SPL {X  -153.706, Y  +316.739, Z    +0.000, E1   +47.523, E3 +314478.356}
SPL {X  -146.106, Y  +300.443, Z    +0.000, E1   +52.765, E3 +314477.975}
SPL {X  -140.816, Y  +291.260, Z    +0.000, E1   +53.766, E3 +314485.658}
SPL {X  -128.440, Y  +273.891, Z    +0.000, E1   +47.966, E3 +314568.745}
ENDSPLINE

SPLINE
SPL {X  -131.798, Y  +278.155, Z    +0.000, E1   +45.574, E3 +314594.372}
SPL {X  -154.181, Y  +317.936, Z    +0.000, E1   +32.662, E3 +314659.709}
SPL {X  -162.537, Y  +346.536, Z    +0.000, E1   +20.123, E3 +314658.929}
SPL {X  -165.197, Y  +366.255, Z    +0.000, E1    +9.700, E3 +314652.725}
SPL {X  -165.621, Y  +375.422, Z    +0.000, E1    +4.067, E3 +314653.125}
SPL {X  -165.650, Y  +379.733, Z    +0.000, E1    +1.160, E3 +314651.431}
SPL {X  -165.650, Y  +383.552, Z    +0.000, E1    -1.868, E3 +314650.681}
SPL {X  -165.650, Y  +387.323, Z    +0.000, E1    -5.609, E3 +314650.497}
SPL {X  -165.650, Y  +392.013, Z    +0.000, E1   -10.856, E3 +314649.515}
SPL {X  -165.650, Y  +398.769, Z    +0.000, E1   -19.304, E3 +314648.126}
SPL {X  -165.650, Y  +410.885, Z    +0.000, E1   -34.864, E3 +314643.802}
SPL {X  -165.650, Y  +448.279, Z    +0.000, E1   -53.294, E3 +314661.647}
SPL {X  -165.650, Y  +465.286, Z    +0.000, E1   -55.209, E3 +314675.499}
SPL {X  -165.650, Y  +513.874, Z    +0.000, E1   -57.683, E3 +314720.307}
ENDSPLINE

SPLINE
SPL {X  -165.650, Y  +513.412, Z    +0.000, E1   -55.245, E3 +314733.903}
SPL {X  -165.650, Y  +495.869, Z    +0.000, E1   -48.812, E3 +314745.204}
ENDSPLINE

SPLINE
SPL {X  -165.650, Y  +502.040, Z    +0.000, E1   -48.856, E3 +314755.948}
SPL {X  -165.650, Y  +507.863, Z    +0.000, E1   -49.013, E3 +314765.368}
SPL {X  -165.650, Y  +512.952, Z    +0.000, E1   -48.898, E3 +314775.145}
SPL {X  -165.650, Y  +519.321, Z    +0.000, E1   -49.041, E3 +314785.613}
SPL {X  -165.650, Y  +524.312, Z    +0.000, E1   -48.855, E3 +314795.638}
SPL {X  -165.650, Y  +530.631, Z    +0.000, E1   -48.990, E3 +314806.098}
SPL {X  -165.650, Y  +536.725, Z    +0.000, E1   -48.843, E3 +314817.849}
SPL {X  -165.650, Y  +542.959, Z    +0.000, E1   -48.923, E3 +314828.464}
SPL {X  -165.650, Y  +548.939, Z    +0.000, E1   -48.968, E3 +314838.858}
SPL {X  -165.650, Y  +553.607, Z    +0.000, E1   -48.716, E3 +314848.676}
SPL {X  -165.650, Y  +562.368, Z    +0.000, E1   -49.014, E3 +314862.736}
SPL {X  -165.650, Y  +570.317, Z    +0.000, E1   -48.893, E3 +314877.479}
SPL {X  -165.650, Y  +577.487, Z    +0.000, E1   -49.001, E3 +314889.587}
SPL {X  -165.650, Y  +581.837, Z    +0.000, E1   -48.612, E3 +314899.621}
SPL {X  -165.650, Y  +588.614, Z    +0.000, E1   -49.053, E3 +314909.138}
SPL {X  -165.650, Y  +593.784, Z    +0.000, E1   -48.711, E3 +314920.424}
SPL {X  -165.650, Y  +600.281, Z    +0.000, E1   -48.957, E3 +314930.526}
SPL {X  -165.650, Y  +606.252, Z    +0.000, E1   -48.984, E3 +314941.060}
SPL {X  -165.650, Y  +612.690, Z    +0.000, E1   -49.044, E3 +314952.088}
SPL {X  -165.650, Y  +617.274, Z    +0.000, E1   -48.670, E3 +314962.537}
SPL {X  -165.650, Y  +624.267, Z    +0.000, E1   -48.953, E3 +314973.349}
SPL {X  -165.650, Y  +632.510, Z    +0.000, E1   -48.976, E3 +314988.104}
SPL {X  -165.650, Y  +641.084, Z    +0.000, E1   -48.892, E3 +315003.746}
SPL {X  -165.650, Y  +648.143, Z    +0.000, E1   -49.033, E3 +315015.415}
SPL {X  -165.650, Y  +652.108, Z    +0.000, E1   -48.593, E3 +315025.100}
SPL {X  -165.650, Y  +658.753, Z    +0.000, E1   -49.107, E3 +315033.925}
SPL {X  -165.650, Y  +663.676, Z    +0.000, E1   -48.809, E3 +315044.471}
SPL {X  -165.650, Y  +669.580, Z    +0.000, E1   -48.844, E3 +315054.810}
SPL {X  -165.650, Y  +675.734, Z    +0.000, E1   -49.021, E3 +315064.716}
SPL {X  -165.552, Y  +681.198, Z    +0.000, E1   -48.804, E3 +315075.796}
SPL {X  -165.221, Y  +687.413, Z    +0.000, E1   -48.790, E3 +315086.968}
SPL {X  -164.785, Y  +692.407, Z    +0.000, E1   -48.653, E3 +315096.683}
SPL {X  -164.074, Y  +698.293, Z    +0.000, E1   -48.857, E3 +315105.967}
SPL {X  -163.489, Y  +702.172, Z    +0.000, E1   -48.443, E3 +315115.284}
SPL {X  -162.217, Y  +709.048, Z    +0.000, E1   -48.328, E3 +315128.424}
SPL {X  -160.800, Y  +715.289, Z    +0.000, E1   -47.964, E3 +315141.432}
SPL {X  -159.392, Y  +720.602, Z    +0.000, E1   -47.892, E3 +315151.343}
SPL {X  -157.947, Y  +725.428, Z    +0.000, E1   -47.498, E3 +315162.082}
SPL {X  -156.133, Y  +730.838, Z    +0.000, E1   -47.305, E3 +315172.799}
SPL {X  -154.870, Y  +734.280, Z    +0.000, E1   -46.924, E3 +315180.803}
SPL {X  -150.529, Y  +744.645, Z    +0.000, E1   -49.720, E3 +315184.076}
SPL {X  -140.987, Y  +762.463, Z    +0.000, E1   -53.922, E3 +315189.108}
SPL {X  -130.133, Y  +777.996, Z    +0.000, E1   -46.969, E3 +315281.533}
ENDSPLINE

SPLINE
SPL {X  -153.839, Y  +736.929, Z    +0.000, E1   -32.772, E3 +315354.604}
SPL {X  -162.700, Y  +706.622, Z    +0.000, E1   -19.657, E3 +315358.897}
SPL {X  -164.822, Y  +692.043, Z    +0.000, E1   -12.043, E3 +315354.536}
SPL {X  -165.501, Y  +682.513, Z    +0.000, E1    -6.586, E3 +315353.230}
SPL {X  -165.645, Y  +676.829, Z    +0.000, E1    -2.974, E3 +315352.573}
SPL {X  -165.650, Y  +673.338, Z    +0.000, E1    -0.547, E3 +315351.743}
SPL {X  -165.650, Y  +670.475, Z    +0.000, E1    +1.794, E3 +315351.666}
SPL {X  -165.650, Y  +667.655, Z    +0.000, E1    +4.420, E3 +315351.462}
SPL {X  -165.650, Y  +664.048, Z    +0.000, E1    +8.230, E3 +315350.839}
SPL {X  -165.650, Y  +658.867, Z    +0.000, E1   +14.313, E3 +315349.303}
SPL {X  -165.650, Y  +650.683, Z    +0.000, E1   +24.801, E3 +315346.738}
SPL {X  -165.650, Y  +640.858, Z    +0.000, E1   +34.904, E3 +315348.482}
SPL {X  -165.650, Y  +633.111, Z    +0.000, E1   +43.522, E3 +315345.376}
SPL {X  -165.650, Y  +594.935, Z    +0.000, E1   +58.150, E3 +315359.976}
SPL {X  -165.650, Y  +579.579, Z    +0.000, E1   +60.394, E3 +315367.860}
SPL {X  -165.650, Y  +536.483, Z    +0.000, E1   +57.139, E3 +315426.142}
ENDSPLINE

SPLINE
SPL {X  -165.650, Y  +561.248, Z    +0.000, E1   +49.247, E3 +315436.832}
ENDSPLINE

SPLINE
SPL {X  -165.650, Y  +558.330, Z    +0.000, E1   +47.867, E3 +315450.556}
SPL {X  -165.650, Y  +550.626, Z    +0.000, E1   +48.045, E3 +315463.566}
SPL {X  -165.650, Y  +545.464, Z    +0.000, E1   +47.668, E3 +315475.435}
SPL {X  -165.650, Y  +535.912, Z    +0.000, E1   +47.888, E3 +315492.021}
SPL {X  -165.650, Y  +526.169, Z    +0.000, E1   +47.853, E3 +315510.201}
SPL {X  -165.650, Y  +517.493, Z    +0.000, E1   +47.895, E3 +315525.949}
SPL {X  -165.650, Y  +511.255, Z    +0.000, E1   +47.920, E3 +315537.238}
SPL {X  -165.650, Y  +507.257, Z    +0.000, E1   +47.748, E3 +315545.619}
SPL {X  -165.650, Y  +501.812, Z    +0.000, E1   +47.738, E3 +315555.903}
SPL {X  -165.650, Y  +493.465, Z    +0.000, E1   +47.959, E3 +315570.073}
SPL {X  -165.650, Y  +486.149, Z    +0.000, E1   +47.831, E3 +315584.348}
SPL {X  -165.650, Y  +479.821, Z    +0.000, E1   +47.727, E3 +315596.622}
SPL {X  -165.650, Y  +472.739, Z    +0.000, E1   +47.923, E3 +315608.641}
SPL {X  -165.650, Y  +465.366, Z    +0.000, E1   +47.775, E3 +315623.221}
SPL {X  -165.650, Y  +456.851, Z    +0.000, E1   +47.856, E3 +315638.527}
SPL {X  -165.650, Y  +449.262, Z    +0.000, E1   +48.080, E3 +315651.093}
SPL {X  -165.650, Y  +436.454, Z    +0.000, E1   +49.483, E3 +315665.800}
SPL {X  -165.650, Y  +428.379, Z    +0.000, E1   +49.373, E3 +315680.396}
SPL {X  -165.650, Y  +423.272, Z    +0.000, E1   +49.176, E3 +315690.532}
SPL {X  -165.650, Y  +416.522, Z    +0.000, E1   +49.338, E3 +315701.510}
SPL {X  -165.650, Y  +410.777, Z    +0.000, E1   +49.173, E3 +315712.562}
SPL {X  -165.650, Y  +405.230, Z    +0.000, E1   +49.266, E3 +315721.766}
SPL {X  -165.650, Y  +398.850, Z    +0.000, E1   +49.279, E3 +315733.057}
SPL {X  -165.650, Y  +391.803, Z    +0.000, E1   +49.319, E3 +315745.095}
SPL {X  -165.650, Y  +386.526, Z    +0.000, E1   +49.193, E3 +315755.184}
SPL {X  -165.649, Y  +378.059, Z    +0.000, E1   +49.283, E3 +315769.727}
SPL {X  -165.292, Y  +367.617, Z    +0.000, E1   +49.239, E3 +315788.492}
SPL {X  -164.692, Y  +360.715, Z    +0.000, E1   +48.960, E3 +315802.026}
SPL {X  -163.908, Y  +354.543, Z    +0.000, E1   +49.169, E3 +315811.717}
SPL {X  -163.052, Y  +349.277, Z    +0.000, E1   +48.680, E3 +315823.823}
SPL {X  -162.125, Y  +344.507, Z    +0.000, E1   +48.543, E3 +315832.962}
SPL {X  -160.947, Y  +339.310, Z    +0.000, E1   +48.561, E3 +315842.071}
SPL {X  -159.499, Y  +333.778, Z    +0.000, E1   +48.145, E3 +315854.184}
SPL {X  -157.957, Y  +328.606, Z    +0.000, E1   +47.890, E3 +315864.608}
SPL {X  -156.095, Y  +323.055, Z    +0.000, E1   +47.566, E3 +315876.292}
SPL {X  -153.706, Y  +316.739, Z    +0.000, E1   +47.523, E3 +315887.446}
SPL {X  -143.727, Y  +296.145, Z    +0.000, E1   +53.260, E3 +315890.590}
SPL {X  -128.440, Y  +273.891, Z    +0.000, E1   +47.966, E3 +315977.836}
ENDSPLINE

SPLINE
SPL {X  -131.798, Y  +278.155, Z    +0.000, E1   +45.574, E3 +316003.463}
SPL {X  -154.181, Y  +317.936, Z    +0.000, E1   +32.662, E3 +316068.800}
SPL {X  -162.537, Y  +346.536, Z    +0.000, E1   +20.123, E3 +316068.020}
SPL {X  -164.610, Y  +359.970, Z    +0.000, E1   +13.118, E3 +316062.887}
SPL {X  -165.367, Y  +368.828, Z    +0.000, E1    +8.137, E3 +316061.339}
SPL {X  -165.621, Y  +375.422, Z    +0.000, E1    +4.067, E3 +316062.216}
SPL {X  -165.650, Y  +380.991, Z    +0.000, E1    +0.306, E3 +316060.228}
SPL {X  -165.650, Y  +384.571, Z    +0.000, E1    -2.883, E3 +316059.667}
SPL {X  -165.650, Y  +388.716, Z    +0.000, E1    -7.003, E3 +316059.176}
SPL {X  -165.650, Y  +396.644, Z    +0.000, E1   -16.434, E3 +316057.795}
SPL {X  -165.650, Y  +407.471, Z    +0.000, E1   -31.017, E3 +316053.376}
SPL {X  -165.650, Y  +414.706, Z    +0.000, E1   -39.242, E3 +316052.352}
SPL {X  -165.650, Y  +446.037, Z    +0.000, E1   -53.739, E3 +316066.957}
SPL {X  -165.650, Y  +454.158, Z    +0.000, E1   -53.343, E3 +316077.309}
SPL {X  -165.650, Y  +513.780, Z    +0.000, E1   -56.183, E3 +316138.106}
ENDSPLINE

SPLINE
SPL {X  -165.650, Y  +495.869, Z    +0.000, E1   -48.812, E3 +316154.295}
ENDSPLINE

SPLINE
SPL {X  -165.650, Y  +502.040, Z    +0.000, E1   -48.856, E3 +316165.039}
SPL {X  -165.650, Y  +507.863, Z    +0.000, E1   -49.013, E3 +316174.459}
SPL {X  -165.650, Y  +512.952, Z    +0.000, E1   -48.898, E3 +316184.236}
SPL {X  -165.650, Y  +519.321, Z    +0.000, E1   -49.041, E3 +316194.704}
SPL {X  -165.650, Y  +524.312, Z    +0.000, E1   -48.855, E3 +316204.729}
SPL {X  -165.650, Y  +532.191, Z    +0.000, E1   -48.944, E3 +316218.397}
SPL {X  -165.650, Y  +541.400, Z    +0.000, E1   -48.945, E3 +316234.772}
SPL {X  -165.650, Y  +548.939, Z    +0.000, E1   -48.968, E3 +316247.949}
SPL {X  -165.650, Y  +553.607, Z    +0.000, E1   -48.716, E3 +316257.767}
SPL {X  -165.650, Y  +562.368, Z    +0.000, E1   -49.014, E3 +316271.827}
SPL {X  -165.650, Y  +570.317, Z    +0.000, E1   -48.893, E3 +316286.570}
SPL {X  -165.650, Y  +577.487, Z    +0.000, E1   -49.001, E3 +316298.678}
SPL {X  -165.650, Y  +581.837, Z    +0.000, E1   -48.612, E3 +316308.712}
SPL {X  -165.650, Y  +588.614, Z    +0.000, E1   -49.053, E3 +316318.229}
SPL {X  -165.650, Y  +593.784, Z    +0.000, E1   -48.711, E3 +316329.515}
SPL {X  -165.650, Y  +600.281, Z    +0.000, E1   -48.957, E3 +316339.617}
SPL {X  -165.650, Y  +606.252, Z    +0.000, E1   -48.984, E3 +316350.150}
SPL {X  -165.650, Y  +612.690, Z    +0.000, E1   -49.044, E3 +316361.179}
SPL {X  -165.650, Y  +617.274, Z    +0.000, E1   -48.670, E3 +316371.628}
SPL {X  -165.650, Y  +624.267, Z    +0.000, E1   -48.953, E3 +316382.440}
SPL {X  -165.650, Y  +632.510, Z    +0.000, E1   -48.976, E3 +316397.195}
SPL {X  -165.650, Y  +641.084, Z    +0.000, E1   -48.892, E3 +316412.837}
SPL {X  -165.650, Y  +648.143, Z    +0.000, E1   -49.033, E3 +316424.506}
SPL {X  -165.650, Y  +655.847, Z    +0.000, E1   -48.917, E3 +316439.124}
SPL {X  -165.650, Y  +663.676, Z    +0.000, E1   -48.809, E3 +316453.562}
SPL {X  -165.650, Y  +669.580, Z    +0.000, E1   -48.844, E3 +316463.901}
SPL {X  -165.650, Y  +675.734, Z    +0.000, E1   -49.021, E3 +316473.807}
SPL {X  -165.552, Y  +681.198, Z    +0.000, E1   -48.804, E3 +316484.887}
SPL {X  -165.221, Y  +687.413, Z    +0.000, E1   -48.790, E3 +316496.059}
SPL {X  -164.785, Y  +692.407, Z    +0.000, E1   -48.653, E3 +316505.774}
SPL {X  -164.074, Y  +698.293, Z    +0.000, E1   -48.857, E3 +316515.058}
SPL {X  -163.489, Y  +702.172, Z    +0.000, E1   -48.443, E3 +316524.375}
SPL {X  -162.217, Y  +709.048, Z    +0.000, E1   -48.328, E3 +316537.515}
SPL {X  -160.800, Y  +715.289, Z    +0.000, E1   -47.964, E3 +316550.523}
SPL {X  -159.392, Y  +720.602, Z    +0.000, E1   -47.892, E3 +316560.434}
SPL {X  -157.947, Y  +725.428, Z    +0.000, E1   -47.498, E3 +316571.173}
SPL {X  -156.133, Y  +730.838, Z    +0.000, E1   -47.305, E3 +316581.890}
SPL {X  -154.870, Y  +734.280, Z    +0.000, E1   -46.924, E3 +316589.894}
SPL {X  -150.529, Y  +744.645, Z    +0.000, E1   -49.720, E3 +316593.167}
SPL {X  -140.987, Y  +762.463, Z    +0.000, E1   -53.922, E3 +316598.199}
SPL {X  -129.526, Y  +778.761, Z    +0.000, E1   -47.396, E3 +316686.262}
ENDSPLINE

SPLINE
SPL {X  -152.848, Y  +739.355, Z    +0.000, E1   -33.672, E3 +316761.831}
SPL {X  -162.700, Y  +706.622, Z    +0.000, E1   -19.657, E3 +316767.988}
SPL {X  -164.822, Y  +692.043, Z    +0.000, E1   -12.043, E3 +316763.626}
SPL {X  -165.501, Y  +682.513, Z    +0.000, E1    -6.586, E3 +316762.321}
SPL {X  -165.650, Y  +674.436, Z    +0.000, E1    -1.443, E3 +316761.096}
SPL {X  -165.650, Y  +670.475, Z    +0.000, E1    +1.794, E3 +316760.757}
SPL {X  -165.650, Y  +667.655, Z    +0.000, E1    +4.420, E3 +316760.553}
SPL {X  -165.650, Y  +664.048, Z    +0.000, E1    +8.230, E3 +316759.930}
SPL {X  -165.650, Y  +658.867, Z    +0.000, E1   +14.313, E3 +316758.394}
SPL {X  -165.650, Y  +650.683, Z    +0.000, E1   +24.801, E3 +316755.829}
SPL {X  -165.650, Y  +640.858, Z    +0.000, E1   +34.904, E3 +316757.572}
SPL {X  -165.650, Y  +633.111, Z    +0.000, E1   +43.522, E3 +316754.467}
SPL {X  -165.650, Y  +594.935, Z    +0.000, E1   +58.150, E3 +316769.066}
SPL {X  -165.650, Y  +579.579, Z    +0.000, E1   +60.394, E3 +316776.951}
SPL {X  -165.650, Y  +536.483, Z    +0.000, E1   +57.139, E3 +316835.233}
ENDSPLINE

SPLINE
SPL {X  -165.650, Y  +561.248, Z    +0.000, E1   +49.247, E3 +316845.923}
ENDSPLINE

SPLINE
SPL {X  -165.650, Y  +558.330, Z    +0.000, E1   +47.867, E3 +316859.647}
SPL {X  -165.650, Y  +550.626, Z    +0.000, E1   +48.045, E3 +316872.657}
SPL {X  -165.650, Y  +545.464, Z    +0.000, E1   +47.668, E3 +316884.526}
SPL {X  -165.650, Y  +535.912, Z    +0.000, E1   +47.888, E3 +316901.111}
SPL {X  -165.650, Y  +526.169, Z    +0.000, E1   +47.853, E3 +316919.292}
SPL {X  -165.650, Y  +517.493, Z    +0.000, E1   +47.895, E3 +316935.039}
SPL {X  -165.650, Y  +511.255, Z    +0.000, E1   +47.920, E3 +316946.328}
SPL {X  -165.650, Y  +507.257, Z    +0.000, E1   +47.748, E3 +316954.710}
SPL {X  -165.650, Y  +501.812, Z    +0.000, E1   +47.738, E3 +316964.994}
SPL {X  -165.650, Y  +494.522, Z    +0.000, E1   +48.055, E3 +316976.521}
SPL {X  -165.650, Y  +489.529, Z    +0.000, E1   +47.849, E3 +316986.974}
SPL {X  -165.650, Y  +484.859, Z    +0.000, E1   +47.688, E3 +316996.544}
SPL {X  -165.650, Y  +477.718, Z    +0.000, E1   +47.870, E3 +317008.879}
SPL {X  -165.650, Y  +469.088, Z    +0.000, E1   +47.982, E3 +317024.098}
SPL {X  -165.650, Y  +464.575, Z    +0.000, E1   +47.451, E3 +317035.512}
SPL {X  -165.650, Y  +456.851, Z    +0.000, E1   +47.856, E3 +317047.618}
SPL {X  -165.650, Y  +449.262, Z    +0.000, E1   +48.080, E3 +317060.184}
SPL {X  -165.650, Y  +436.765, Z    +0.000, E1   +49.819, E3 +317072.083}
SPL {X  -165.650, Y  +430.891, Z    +0.000, E1   +49.130, E3 +317086.585}
SPL {X  -165.650, Y  +423.272, Z    +0.000, E1   +49.176, E3 +317099.623}
SPL {X  -165.650, Y  +416.522, Z    +0.000, E1   +49.338, E3 +317110.601}
SPL {X  -165.650, Y  +408.142, Z    +0.000, E1   +49.261, E3 +317125.962}
SPL {X  -165.650, Y  +400.266, Z    +0.000, E1   +49.362, E3 +317139.023}
SPL {X  -165.650, Y  +393.708, Z    +0.000, E1   +49.252, E3 +317151.330}
SPL {X  -165.650, Y  +384.475, Z    +0.000, E1   +49.187, E3 +317168.128}
SPL {X  -165.626, Y  +375.686, Z    +0.000, E1   +49.367, E3 +317182.345}
SPL {X  -165.370, Y  +368.879, Z    +0.000, E1   +49.286, E3 +317194.899}
SPL {X  -164.828, Y  +362.023, Z    +0.000, E1   +48.964, E3 +317208.860}
SPL {X  -164.139, Y  +356.180, Z    +0.000, E1   +49.110, E3 +317218.210}
SPL {X  -163.224, Y  +350.255, Z    +0.000, E1   +48.882, E3 +317230.205}
SPL {X  -162.125, Y  +344.507, Z    +0.000, E1   +48.543, E3 +317242.053}
SPL {X  -160.947, Y  +339.310, Z    +0.000, E1   +48.561, E3 +317251.162}
SPL {X  -159.499, Y  +333.778, Z    +0.000, E1   +48.145, E3 +317263.275}
SPL {X  -157.957, Y  +328.606, Z    +0.000, E1   +47.890, E3 +317273.699}
SPL {X  -156.095, Y  +323.055, Z    +0.000, E1   +47.566, E3 +317285.383}
SPL {X  -153.706, Y  +316.739, Z    +0.000, E1   +47.523, E3 +317296.537}
SPL {X  -143.727, Y  +296.145, Z    +0.000, E1   +53.260, E3 +317299.681}
SPL {X  -128.440, Y  +273.891, Z    +0.000, E1   +47.966, E3 +317386.927}
ENDSPLINE

SPLINE
SPL {X  -131.798, Y  +278.155, Z    +0.000, E1   +45.574, E3 +317412.554}
SPL {X  -154.181, Y  +317.936, Z    +0.000, E1   +32.662, E3 +317477.891}
SPL {X  -162.537, Y  +346.536, Z    +0.000, E1   +20.123, E3 +317477.111}
SPL {X  -165.197, Y  +366.255, Z    +0.000, E1    +9.700, E3 +317470.906}
SPL {X  -165.621, Y  +375.422, Z    +0.000, E1    +4.067, E3 +317471.307}
SPL {X  -165.650, Y  +379.733, Z    +0.000, E1    +1.160, E3 +317469.613}
SPL {X  -165.650, Y  +383.552, Z    +0.000, E1    -1.868, E3 +317468.863}
SPL {X  -165.650, Y  +387.323, Z    +0.000, E1    -5.609, E3 +317468.679}
SPL {X  -165.650, Y  +392.013, Z    +0.000, E1   -10.856, E3 +317467.696}
SPL {X  -165.650, Y  +398.769, Z    +0.000, E1   -19.304, E3 +317466.308}
SPL {X  -165.650, Y  +410.885, Z    +0.000, E1   -34.864, E3 +317461.984}
SPL {X  -165.650, Y  +446.037, Z    +0.000, E1   -53.739, E3 +317476.048}
SPL {X  -165.650, Y  +454.158, Z    +0.000, E1   -53.343, E3 +317486.400}
SPL {X  -165.650, Y  +513.780, Z    +0.000, E1   -56.183, E3 +317547.197}
ENDSPLINE

SPLINE
SPL {X  -165.650, Y  +495.869, Z    +0.000, E1   -48.812, E3 +317563.386}
ENDSPLINE

SPLINE
SPL {X  -165.650, Y  +504.906, Z    +0.000, E1   -48.979, E3 +317578.705}
SPL {X  -165.650, Y  +512.952, Z    +0.000, E1   -48.898, E3 +317593.327}
SPL {X  -165.650, Y  +519.321, Z    +0.000, E1   -49.041, E3 +317603.795}
SPL {X  -165.650, Y  +524.312, Z    +0.000, E1   -48.855, E3 +317613.820}
SPL {X  -165.650, Y  +530.631, Z    +0.000, E1   -48.990, E3 +317624.280}
SPL {X  -165.650, Y  +536.725, Z    +0.000, E1   -48.843, E3 +317636.031}
SPL {X  -165.650, Y  +542.959, Z    +0.000, E1   -48.923, E3 +317646.646}
SPL {X  -165.650, Y  +548.939, Z    +0.000, E1   -48.968, E3 +317657.040}
SPL {X  -165.650, Y  +553.607, Z    +0.000, E1   -48.716, E3 +317666.858}
SPL {X  -165.650, Y  +562.368, Z    +0.000, E1   -49.014, E3 +317680.918}
SPL {X  -165.650, Y  +570.317, Z    +0.000, E1   -48.893, E3 +317695.661}
SPL {X  -165.650, Y  +577.487, Z    +0.000, E1   -49.001, E3 +317707.769}
SPL {X  -165.650, Y  +581.837, Z    +0.000, E1   -48.612, E3 +317717.802}
SPL {X  -165.650, Y  +588.614, Z    +0.000, E1   -49.053, E3 +317727.320}
SPL {X  -165.650, Y  +593.784, Z    +0.000, E1   -48.711, E3 +317738.606}
SPL {X  -165.650, Y  +600.281, Z    +0.000, E1   -48.957, E3 +317748.708}
SPL {X  -165.650, Y  +606.252, Z    +0.000, E1   -48.984, E3 +317759.241}
SPL {X  -165.650, Y  +612.690, Z    +0.000, E1   -49.044, E3 +317770.270}
SPL {X  -165.650, Y  +617.274, Z    +0.000, E1   -48.670, E3 +317780.719}
SPL {X  -165.650, Y  +624.267, Z    +0.000, E1   -48.953, E3 +317791.531}
SPL {X  -165.650, Y  +632.510, Z    +0.000, E1   -48.976, E3 +317806.286}
SPL {X  -165.650, Y  +641.084, Z    +0.000, E1   -48.892, E3 +317821.928}
SPL {X  -165.650, Y  +648.143, Z    +0.000, E1   -49.033, E3 +317833.597}
SPL {X  -165.650, Y  +655.847, Z    +0.000, E1   -48.917, E3 +317848.215}
SPL {X  -165.650, Y  +663.676, Z    +0.000, E1   -48.809, E3 +317862.653}
SPL {X  -165.650, Y  +669.580, Z    +0.000, E1   -48.844, E3 +317872.991}
SPL {X  -165.650, Y  +675.734, Z    +0.000, E1   -49.021, E3 +317882.898}
SPL {X  -165.552, Y  +681.198, Z    +0.000, E1   -48.804, E3 +317893.978}
SPL {X  -165.221, Y  +687.413, Z    +0.000, E1   -48.790, E3 +317905.150}
SPL {X  -164.785, Y  +692.407, Z    +0.000, E1   -48.653, E3 +317914.865}
SPL {X  -164.074, Y  +698.293, Z    +0.000, E1   -48.857, E3 +317924.149}
SPL {X  -163.489, Y  +702.172, Z    +0.000, E1   -48.443, E3 +317933.466}
SPL {X  -162.217, Y  +709.048, Z    +0.000, E1   -48.328, E3 +317946.606}
SPL {X  -160.800, Y  +715.289, Z    +0.000, E1   -47.964, E3 +317959.613}
SPL {X  -159.392, Y  +720.602, Z    +0.000, E1   -47.892, E3 +317969.525}
SPL {X  -157.947, Y  +725.428, Z    +0.000, E1   -47.498, E3 +317980.264}
SPL {X  -156.133, Y  +730.838, Z    +0.000, E1   -47.305, E3 +317990.981}
SPL {X  -153.862, Y  +736.871, Z    +0.000, E1   -47.425, E3 +318000.968}
SPL {X  -143.211, Y  +758.749, Z    +0.000, E1   -53.445, E3 +318004.611}
SPL {X  -130.133, Y  +777.996, Z    +0.000, E1   -46.969, E3 +318099.714}
ENDSPLINE

SPLINE
SPL {X  -153.839, Y  +736.929, Z    +0.000, E1   -32.772, E3 +318172.786}
SPL {X  -162.700, Y  +706.622, Z    +0.000, E1   -19.657, E3 +318177.079}
SPL {X  -164.822, Y  +692.043, Z    +0.000, E1   -12.043, E3 +318172.717}
SPL {X  -165.501, Y  +682.513, Z    +0.000, E1    -6.586, E3 +318171.412}
SPL {X  -165.650, Y  +674.436, Z    +0.000, E1    -1.443, E3 +318170.187}
SPL {X  -165.650, Y  +669.008, Z    +0.000, E1    +2.993, E3 +318169.742}
SPL {X  -165.650, Y  +664.048, Z    +0.000, E1    +8.230, E3 +318169.021}
SPL {X  -165.650, Y  +658.867, Z    +0.000, E1   +14.313, E3 +318167.485}
SPL {X  -165.650, Y  +650.683, Z    +0.000, E1   +24.801, E3 +318164.920}
SPL {X  -165.650, Y  +636.402, Z    +0.000, E1   +39.824, E3 +318164.883}
SPL {X  -165.650, Y  +586.376, Z    +0.000, E1   +59.481, E3 +318182.555}
SPL {X  -165.650, Y  +558.853, Z    +0.000, E1   +50.142, E3 +318254.025}
SPL {X  -165.650, Y  +558.330, Z    +0.000, E1   +47.867, E3 +318268.738}
SPL {X  -165.650, Y  +550.626, Z    +0.000, E1   +48.045, E3 +318281.748}
SPL {X  -165.650, Y  +545.464, Z    +0.000, E1   +47.668, E3 +318293.617}
SPL {X  -165.650, Y  +537.837, Z    +0.000, E1   +47.880, E3 +318306.494}
SPL {X  -165.650, Y  +530.616, Z    +0.000, E1   +47.886, E3 +318319.860}
SPL {X  -165.650, Y  +524.679, Z    +0.000, E1   +47.721, E3 +318331.752}
SPL {X  -165.650, Y  +517.493, Z    +0.000, E1   +47.895, E3 +318344.130}
SPL {X  -165.650, Y  +509.413, Z    +0.000, E1   +47.884, E3 +318359.210}
SPL {X  -165.650, Y  +501.812, Z    +0.000, E1   +47.738, E3 +318374.084}
SPL {X  -165.650, Y  +494.522, Z    +0.000, E1   +48.055, E3 +318385.611}
SPL {X  -165.650, Y  +489.529, Z    +0.000, E1   +47.849, E3 +318396.065}
SPL {X  -165.650, Y  +481.894, Z    +0.000, E1   +47.756, E3 +318410.966}
SPL {X  -165.650, Y  +472.739, Z    +0.000, E1   +47.923, E3 +318426.823}
SPL {X  -165.650, Y  +465.366, Z    +0.000, E1   +47.775, E3 +318441.402}
SPL {X  -165.650, Y  +457.811, Z    +0.000, E1   +47.987, E3 +318454.019}
SPL {X  -165.650, Y  +451.187, Z    +0.000, E1   +47.917, E3 +318466.763}
SPL {X  -165.650, Y  +436.765, Z    +0.000, E1   +49.819, E3 +318481.174}
SPL {X  -165.650, Y  +430.891, Z    +0.000, E1   +49.130, E3 +318495.676}
SPL {X  -165.650, Y  +423.272, Z    +0.000, E1   +49.176, E3 +318508.714}
SPL {X  -165.650, Y  +416.522, Z    +0.000, E1   +49.338, E3 +318519.692}
SPL {X  -165.650, Y  +410.777, Z    +0.000, E1   +49.173, E3 +318530.744}
SPL {X  -165.650, Y  +405.230, Z    +0.000, E1   +49.266, E3 +318539.948}
SPL {X  -165.650, Y  +398.850, Z    +0.000, E1   +49.279, E3 +318551.239}
SPL {X  -165.650, Y  +391.803, Z    +0.000, E1   +49.319, E3 +318563.277}
SPL {X  -165.650, Y  +386.526, Z    +0.000, E1   +49.193, E3 +318573.366}
SPL {X  -165.649, Y  +378.059, Z    +0.000, E1   +49.283, E3 +318587.909}
SPL {X  -165.292, Y  +367.617, Z    +0.000, E1   +49.239, E3 +318606.674}
SPL {X  -164.692, Y  +360.715, Z    +0.000, E1   +48.960, E3 +318620.208}
SPL {X  -163.908, Y  +354.543, Z    +0.000, E1   +49.169, E3 +318629.899}
SPL {X  -163.052, Y  +349.277, Z    +0.000, E1   +48.680, E3 +318642.005}
SPL {X  -162.125, Y  +344.507, Z    +0.000, E1   +48.543, E3 +318651.144}
SPL {X  -160.947, Y  +339.310, Z    +0.000, E1   +48.561, E3 +318660.253}
SPL {X  -159.499, Y  +333.778, Z    +0.000, E1   +48.145, E3 +318672.366}
SPL {X  -157.957, Y  +328.606, Z    +0.000, E1   +47.890, E3 +318682.790}
SPL {X  -156.095, Y  +323.055, Z    +0.000, E1   +47.566, E3 +318694.474}
SPL {X  -153.706, Y  +316.739, Z    +0.000, E1   +47.523, E3 +318705.628}
SPL {X  -143.727, Y  +296.145, Z    +0.000, E1   +53.260, E3 +318708.772}
SPL {X  -128.440, Y  +273.891, Z    +0.000, E1   +47.966, E3 +318796.018}
ENDSPLINE

SPLINE
SPL {X  -131.798, Y  +278.155, Z    +0.000, E1   +45.574, E3 +318821.645}
SPL {X  -154.181, Y  +317.936, Z    +0.000, E1   +32.662, E3 +318886.981}
SPL {X  -162.537, Y  +346.536, Z    +0.000, E1   +20.123, E3 +318886.202}
SPL {X  -165.197, Y  +366.255, Z    +0.000, E1    +9.700, E3 +318879.997}
SPL {X  -165.621, Y  +375.422, Z    +0.000, E1    +4.067, E3 +318880.398}
SPL {X  -165.650, Y  +379.733, Z    +0.000, E1    +1.160, E3 +318878.704}
SPL {X  -165.650, Y  +383.552, Z    +0.000, E1    -1.868, E3 +318877.954}
SPL {X  -165.650, Y  +387.323, Z    +0.000, E1    -5.609, E3 +318877.770}
SPL {X  -165.650, Y  +392.013, Z    +0.000, E1   -10.856, E3 +318876.787}
SPL {X  -165.650, Y  +398.769, Z    +0.000, E1   -19.304, E3 +318875.399}
SPL {X  -165.650, Y  +410.885, Z    +0.000, E1   -34.864, E3 +318871.075}
SPL {X  -165.650, Y  +448.279, Z    +0.000, E1   -53.294, E3 +318888.920}
SPL {X  -165.650, Y  +465.286, Z    +0.000, E1   -55.209, E3 +318902.771}
SPL {X  -165.650, Y  +513.780, Z    +0.000, E1   -56.183, E3 +318956.288}
ENDSPLINE

SPLINE
SPL {X  -165.650, Y  +495.869, Z    +0.000, E1   -48.812, E3 +318972.477}
ENDSPLINE

SPLINE
SPL {X  -165.650, Y  +504.906, Z    +0.000, E1   -48.979, E3 +318987.796}
SPL {X  -165.650, Y  +512.952, Z    +0.000, E1   -48.898, E3 +319002.418}
SPL {X  -165.650, Y  +519.321, Z    +0.000, E1   -49.041, E3 +319012.886}
SPL {X  -165.650, Y  +524.312, Z    +0.000, E1   -48.855, E3 +319022.911}
SPL {X  -165.650, Y  +530.631, Z    +0.000, E1   -48.990, E3 +319033.371}
SPL {X  -165.650, Y  +536.725, Z    +0.000, E1   -48.843, E3 +319045.122}
SPL {X  -165.650, Y  +542.959, Z    +0.000, E1   -48.923, E3 +319055.737}
SPL {X  -165.650, Y  +548.939, Z    +0.000, E1   -48.968, E3 +319066.131}
SPL {X  -165.650, Y  +553.607, Z    +0.000, E1   -48.716, E3 +319075.949}
SPL {X  -165.650, Y  +562.368, Z    +0.000, E1   -49.014, E3 +319090.009}
SPL {X  -165.650, Y  +570.317, Z    +0.000, E1   -48.893, E3 +319104.752}
SPL {X  -165.650, Y  +577.487, Z    +0.000, E1   -49.001, E3 +319116.860}
SPL {X  -165.650, Y  +581.837, Z    +0.000, E1   -48.612, E3 +319126.893}
SPL {X  -165.650, Y  +588.614, Z    +0.000, E1   -49.053, E3 +319136.411}
SPL {X  -165.650, Y  +593.784, Z    +0.000, E1   -48.711, E3 +319147.696}
SPL {X  -165.650, Y  +600.281, Z    +0.000, E1   -48.957, E3 +319157.799}
SPL {X  -165.650, Y  +606.252, Z    +0.000, E1   -48.984, E3 +319168.332}
SPL {X  -165.650, Y  +612.690, Z    +0.000, E1   -49.044, E3 +319179.361}
SPL {X  -165.650, Y  +617.274, Z    +0.000, E1   -48.670, E3 +319189.810}
SPL {X  -165.650, Y  +624.267, Z    +0.000, E1   -48.953, E3 +319200.622}
SPL {X  -165.650, Y  +632.510, Z    +0.000, E1   -48.976, E3 +319215.377}
SPL {X  -165.650, Y  +641.084, Z    +0.000, E1   -48.892, E3 +319231.019}
SPL {X  -165.650, Y  +648.143, Z    +0.000, E1   -49.033, E3 +319242.688}
SPL {X  -165.650, Y  +655.847, Z    +0.000, E1   -48.917, E3 +319257.306}
SPL {X  -165.650, Y  +663.676, Z    +0.000, E1   -48.809, E3 +319271.744}
SPL {X  -165.650, Y  +669.580, Z    +0.000, E1   -48.844, E3 +319282.082}
SPL {X  -165.650, Y  +675.734, Z    +0.000, E1   -49.021, E3 +319291.989}
SPL {X  -165.552, Y  +681.198, Z    +0.000, E1   -48.804, E3 +319303.069}
SPL {X  -165.221, Y  +687.413, Z    +0.000, E1   -48.790, E3 +319314.240}
SPL {X  -164.785, Y  +692.407, Z    +0.000, E1   -48.653, E3 +319323.956}
SPL {X  -164.074, Y  +698.293, Z    +0.000, E1   -48.857, E3 +319333.240}
SPL {X  -163.489, Y  +702.172, Z    +0.000, E1   -48.443, E3 +319342.557}
SPL {X  -162.671, Y  +706.776, Z    +0.000, E1   -48.273, E3 +319351.776}
SPL {X  -161.177, Y  +713.734, Z    +0.000, E1   -48.156, E3 +319365.062}
SPL {X  -159.392, Y  +720.602, Z    +0.000, E1   -47.892, E3 +319378.616}
SPL {X  -157.947, Y  +725.428, Z    +0.000, E1   -47.498, E3 +319389.355}
SPL {X  -155.696, Y  +732.057, Z    +0.000, E1   -47.224, E3 +319402.832}
SPL {X  -152.475, Y  +740.240, Z    +0.000, E1   -48.059, E3 +319412.661}
SPL {X  -143.211, Y  +758.749, Z    +0.000, E1   -53.445, E3 +319413.702}
SPL {X  -129.526, Y  +778.761, Z    +0.000, E1   -47.396, E3 +319504.444}
ENDSPLINE

SPLINE
SPL {X  -152.848, Y  +739.355, Z    +0.000, E1   -33.672, E3 +319580.013}
SPL {X  -162.700, Y  +706.622, Z    +0.000, E1   -19.657, E3 +319586.170}
SPL {X  -164.822, Y  +692.043, Z    +0.000, E1   -12.043, E3 +319581.808}
SPL {X  -165.501, Y  +682.513, Z    +0.000, E1    -6.586, E3 +319580.503}
SPL {X  -165.650, Y  +674.436, Z    +0.000, E1    -1.443, E3 +319579.278}
SPL {X  -165.650, Y  +669.008, Z    +0.000, E1    +2.993, E3 +319578.833}
SPL {X  -165.650, Y  +664.048, Z    +0.000, E1    +8.230, E3 +319578.112}
SPL {X  -165.650, Y  +658.867, Z    +0.000, E1   +14.313, E3 +319576.576}
SPL {X  -165.650, Y  +650.683, Z    +0.000, E1   +24.801, E3 +319574.011}
SPL {X  -165.650, Y  +640.858, Z    +0.000, E1   +34.904, E3 +319575.754}
SPL {X  -165.650, Y  +633.111, Z    +0.000, E1   +43.522, E3 +319572.649}
SPL {X  -165.650, Y  +586.376, Z    +0.000, E1   +59.481, E3 +319591.646}
SPL {X  -165.650, Y  +554.310, Z    +0.000, E1   +51.914, E3 +319659.690}
ENDSPLINE

SPLINE
SPL {X  -165.650, Y  +561.648, Z    +0.000, E1   +48.058, E3 +319670.507}
ENDSPLINE

